// TwinCAT 3 PLC project MotorControl
// ProgramVersion: 3.1.4024.0
// libraries:
//   Tc2_ModbusRTU, * (Beckhoff Automation GmbH)
//   Tc2_Standard, * (Beckhoff Automation GmbH)
//   Tc2_System, * (Beckhoff Automation GmbH)
//   Tc3_Module, * (Beckhoff Automation GmbH)
// project tree:
//   DUTs/ E_Command.TcDUT, E_InverterControlWord.TcDUT, E_InverterStatusWord.TcTLEO, E_InverterError.TcTLEO, E_StateDevice.TcTLEO, ST_Inverter.TcDUT, ST_WorkTime.TcDUT
//   DUTs/Fermentation/ ST_LevelSens.TcDUT, ST_MccRev.TcDUT, ST_PhSens.TcDUT, ST_PressureSens.TcDUT, ST_TempSens.TcDUT
//   GVLs/GVL.FermentationProcess/ Fermentation_001.TcGVL
//   GVLs/ GVL.TcGVL, Itf.TcGVL, Param.TcGVL
//   / PlcTask.TcTTO
//   POUs/Abstraction/ FB_MotorControl.TcPOU, FB_MotorControlInverter.TcPOU, FB_MotorControlReverse.TcPOU
//   POUs/Devices/ Button.TcPOU, Button_1.TcPOU, Contactor.TcPOU, ContactorReverse.TcPOU, NumberEdit.TcPOU, Label.TcPOU, Led.TcPOU, TermFuse.TcPOU
//   POUs/Devices/ITFs/ I_Button.TcIO
//   POUs/Devices/Modbus/ FB_InverterOperation.TcPOU
//   POUs/Implementation/ FB_Drive.TcPOU, FB_DriveInverter.TcPOU, FB_DriveReverse.TcPOU
//   POUs/Implementation/ITFs/ I_Drive.TcIO, I_DriveInverter.TcIO, I_DriveReverse.TcIO
//   POUs/ MAIN.TcPOU, mergeIO.TcPOU
//   POUs/Process/ FermentationProcess_001.TcPOU
//   POUs/Scaling/ FB_Scaling.TcPOU
// (motion and I/O tree: see PLC project mcc)
// real-time tasks:
//   TASK PlcTask2: cycle T#10ms, priority 22, ADS port 352
// variable links:

CONFIGURATION MotorControl
    RESOURCE PLC ON TwinCAT3
        TASK PlcTask(INTERVAL := T#10ms, PRIORITY := 22);
        PROGRAM MAIN WITH PlcTask : MAIN;
    END_RESOURCE
END_CONFIGURATION

// ---- DUTs/E_Command.TcDUT
//{attribute 'qualified_only'}
{attribute 'strict'}
TYPE E_Command :
(
	 eReady, 
	 eFwd, 
	 eRev,
	 eResetInv  
	 
); // domyślna inicjalizacja wszystkich E_ATVCommand Variables na WORD
END_TYPE

// ---- DUTs/E_InverterControlWord.TcDUT
//{attribute 'qualified_only'}
{attribute 'strict'}
TYPE E_InverterControlWord :
(
	 eShutDown         := 16#0006,  //State 2 - Shutdown command -final operating state -> Ready to switch on 
	 eSwitchOn         := 16#0007,  //State 3 - Switch On  command - final operating state -> Switched On Its the same command Disable Operation
	 eEnableOperation  := 16#000F,	//State 4 - Enable Operation - final operating state -> Operation enabled (napęd pracuej do przodu)  
	 eReverseOperation := 16#080F,  //State 4 - Enable Operation Reverse - final operating state -> Operation enabled (napęd pracuej do tyłu)
	 eFaultReset       := 16#0080   //State 5 - Error reset - final operating state -> Ready to switch on 
 	 
)WORD;
END_TYPE

// ---- DUTs/E_InverterStatusWord.TcTLEO
//{attribute 'qualified_only'}
{attribute 'strict'}
TYPE E_InverterStatusWord : // State WORD of ATV Inverter ETA Masked By 0x006f H
(
	eFaultAfterOperation   := 16#0008,	// wykryto błąd po stanie operacyjnym (falownik pracował i nastąpił błąd pracy) po operacji Quick Stop Active przejscie do stanu - 6 falownika
	eFaultDrive            := 16#0028,	// błąd komunikacja Modbus przerwana i nieaktywna SLF1
	eSwitchOnDisabled	   := 16#0040,	// Stan po udanym resecie błędu komunikacji LCD - nSE
	eReadyToSwitchOn       := 16#0021,	// Stan po ustawieniu gotowości Inverta komendą eReady = 14
	eSwitchedOn            := 16#0023,  // Stan po ustawieniu komendy eFwd = 15 lub eRev = 2063 gdy jest zerowa prędkośc zadana speed = 0 
	eOperationEnabled      := 16#0027   // Stan gdy napęd pracuje w kierunku do przodu i do tyłu i osiagnał predkosc zadaną
		
)WORD;
END_TYPE
//  eFaultAfterOperation = '16#0008'
//  eFaultDrive = '16#0028'
//  eSwitchOnDisabled = '16#0040'
//  eReadyToSwitchOn = '16#0021'
//  eSwitchedOn = '16#0023'
//  eOperationEnabled = '16#0027'

// ---- DUTs/E_InverterError.TcTLEO
{attribute 'qualified_only'}
{attribute 'strict'}
TYPE E_InverterError :
(
	nOF := 0,
	InF := 1,
	CFF := 3,
	CFI := 4,
	SLF1:= 5, 
	EPF1:= 8,
	OCF := 9,
	CrF1:= 10,
	OHF := 16,
	OLF := 17,
	ObF := 18,
	OSF := 19,
	OPF1:= 20,
	PHF := 21,
	USF := 22,
	SCF1:= 23,
	SOF := 24,
	tnF := 25,
	InF1:= 26,
	InF2:= 27,
	InF3:= 28,
	InF4:= 29,
	SCF3:= 32,
	OPF2:= 33,
	SLF2:= 42,
	SLF3:= 45,
	InF9:= 51,
	InFb:= 53,
	tJF := 54,
	SCF4:= 55,
	SCF5:= 56,
	InFE:= 69, 
	CFI2:= 77,
	ULF := 100,
	OLC := 101,
	SPIF:= 102,
	LFF1:= 106
	
)WORD;
END_TYPE

// ---- DUTs/E_StateDevice.TcTLEO
//{attribute 'qualified_only'}
{attribute 'strict'}
TYPE E_StateDevice :
(
	eOn       := 0,
	eOff      := 1,
	eForward  := 2,
	eReverse  := 3,
	eReset    := 4,
	eFault    := 5,
	eAuto     := 6
);
END_TYPE

// ---- DUTs/Fermentation/ST_LevelSens.TcDUT
{attribute 'OPC.UA.DA' := '2'}
{attribute 'OPC.UA.DA.StructuredType' := '1'}

TYPE ST_LevelSens :
STRUCT
	
	rRawLevelValue AT%I* : INT;	 // raw value from measure instruments
	rLevelValue  		 : REAL;  // value from fermentation tank Level sensor	

END_STRUCT
END_TYPE

// ---- DUTs/Fermentation/ST_MccRev.TcDUT
{attribute 'OPC.UA.DA' := '2'}
{attribute 'OPC.UA.DA.StructuredType' := '1'}
TYPE ST_MccRev :
STRUCT

	bAutoButton  	   : BOOL;  // SCADA button Auto/manual Command
	bForwardButton     : BOOL;  // SCADA button Forward drive Command
	bReverseButton	   : BOOL;  // SCADA button Reverse drive Command
	bTermFuse    AT%I* : BOOL;  // Term Fuse state from psyhical input
	bContactor   AT%Q* : BOOL;  // Contactor state from psyhical output
	udHours   		   : UDINT; // Work Time Counter - hours nonvolatile memory register
	uMinutes	   	   : UINT;  // Work Time Counter - minuts nonvolatile memory register
	uSeconds           : UINT;  // Work Time Counter - seconds nonvolatile memory register
  	sStatus	           : T_MaxString; // Motor Status string
	sState 	           : T_MaxString; // Motor State string		

END_STRUCT
END_TYPE

// ---- DUTs/Fermentation/ST_PhSens.TcDUT
{attribute 'OPC.UA.DA' := '2'}
{attribute 'OPC.UA.DA.StructuredType' := '1'}

TYPE ST_PhSens :
STRUCT
	
	rRawPhValue AT%I* : INT;	 // raw value from measure instruments
	rPhValue  		  : REAL;    // value from fermentation tank Ph sensor		

END_STRUCT
END_TYPE

// ---- DUTs/Fermentation/ST_PressureSens.TcDUT
{attribute 'OPC.UA.DA' := '2'}
{attribute 'OPC.UA.DA.StructuredType' := '1'}
TYPE ST_PressureSens :
STRUCT
	
	rRawPressureValue AT%I* : INT;	   // raw value from measure instruments
	rPressureValue  		: REAL;    // value from fermentation tank Pressure sensor	

END_STRUCT
END_TYPE

// ---- DUTs/Fermentation/ST_TempSens.TcDUT
{attribute 'OPC.UA.DA' := '2'}
{attribute 'OPC.UA.DA.StructuredType' := '1'}
TYPE ST_TempSens :
STRUCT
	
	rRawTempValue AT%I* : INT;	 // raw value from measure instruments
	rTempValue  		: REAL;  // value from fermentation tank temperature sensor	

END_STRUCT
END_TYPE

// ---- DUTs/ST_Inverter.TcDUT
TYPE ST_Inverter :
STRUCT
	bDeviceId         : BYTE;
	wStatus	          : E_InverterStatusWord;
	eControl          : E_InverterControlWord;
	errorInv  		  : E_InverterError;           // AVT inverter Error
	sErrorDescription : T_MaxString;
	rSpeed	          : WORD;	
	errorMdb          : MODBUS_ERRORS;  // Modbus Communications error		
END_STRUCT
END_TYPE

// ---- DUTs/ST_WorkTime.TcDUT
TYPE ST_WorkTime :
STRUCT
	hours	: UDINT;
	minuts	: UINT;
	seconds	: UINT;
END_STRUCT
END_TYPE

// ---- GVLs/GVL.FermentationProcess/Fermentation_001.TcGVL
{attribute 'qualified_only'}
VAR_GLOBAL
	
	//**************************** Reverse Motor ***************************************************************
	
	{attribute 'OPC.UA.DA' := '1'}
	{attribute 'OPC.UA.DA.StructuredType' := '1'}
	{attribute 'OPC.UA.DA.Description' := 'MccRev (structured) type '} 
	MccRev_001 : ST_MccRev;
	
	{attribute 'OPC.UA.DA' := '1'}
	{attribute 'OPC.UA.DA.StructuredType' := '1'}
	{attribute 'OPC.UA.DA.Description' := 'MccRev (structured) type '} 
	MccRev_002 : ST_MccRev;
	
	{attribute 'OPC.UA.DA' := '1'}
	{attribute 'OPC.UA.DA.StructuredType' := '1'}
	{attribute 'OPC.UA.DA.Description' := 'MccRev (structured) type '} 
	MccRev_003 : ST_MccRev;
	
	{attribute 'OPC.UA.DA' := '1'}
	{attribute 'OPC.UA.DA.StructuredType' := '1'}
	{attribute 'OPC.UA.DA.Description' := 'MccRev (structured) type '} 
	MccRev_004 : ST_MccRev;
	
	{attribute 'OPC.UA.DA' := '1'}
	{attribute 'OPC.UA.DA.StructuredType' := '1'}
	{attribute 'OPC.UA.DA.Description' := 'MccRev (structured) type '} 
	MccRev_005 : ST_MccRev;
	
	{attribute 'OPC.UA.DA' := '1'}
	{attribute 'OPC.UA.DA.StructuredType' := '1'}
	{attribute 'OPC.UA.DA.Description' := 'MccRev (structured) type '} 
	MccRev_006 : ST_MccRev;
	
	{attribute 'OPC.UA.DA' := '1'}
	{attribute 'OPC.UA.DA.StructuredType' := '1'}
	{attribute 'OPC.UA.DA.Description' := 'MccRev (structured) type '} 
	MccRev_007 : ST_MccRev;
	
	{attribute 'OPC.UA.DA' := '1'}
	{attribute 'OPC.UA.DA.StructuredType' := '1'}
	{attribute 'OPC.UA.DA.Description' := 'MccRev (structured) type '} 
	MccRev_008 : ST_MccRev;
	
	{attribute 'OPC.UA.DA' := '1'}
	{attribute 'OPC.UA.DA.StructuredType' := '1'}
	{attribute 'OPC.UA.DA.Description' := 'MccRev (structured) type '} 
	MccRev_009 : ST_MccRev;
	
	{attribute 'OPC.UA.DA' := '1'}
	{attribute 'OPC.UA.DA.StructuredType' := '1'}
	{attribute 'OPC.UA.DA.Description' := 'MccRev (structured) type '} 
	MccRev_010 : ST_MccRev;
	
	{attribute 'OPC.UA.DA' := '1'}
	{attribute 'OPC.UA.DA.StructuredType' := '1'}
	{attribute 'OPC.UA.DA.Description' := 'MccRev (structured) type '} 
	MccRev_011 : ST_MccRev;
	
	
	{attribute 'OPC.UA.DA' := '1'}
	{attribute 'OPC.UA.DA.StructuredType' := '1'}
	{attribute 'OPC.UA.DA.Description' := 'MccRev (structured) type '} 
	MccRev_012 : ST_MccRev;
	
	
	{attribute 'OPC.UA.DA' := '1'}
	{attribute 'OPC.UA.DA.StructuredType' := '1'}
	{attribute 'OPC.UA.DA.Description' := 'MccRev (structured) type '} 
	MccRev_013 : ST_MccRev;
	
	{attribute 'OPC.UA.DA' := '1'}
	{attribute 'OPC.UA.DA.StructuredType' := '1'}
	{attribute 'OPC.UA.DA.Description' := 'MccRev (structured) type '} 
	MccRev_014 : ST_MccRev;
	
	
	{attribute 'OPC.UA.DA' := '1'}
	{attribute 'OPC.UA.DA.StructuredType' := '1'}
	{attribute 'OPC.UA.DA.Description' := 'MccRev (structured) type '} 
	MccRev_015 : ST_MccRev;
	
	
	{attribute 'OPC.UA.DA' := '1'}
	{attribute 'OPC.UA.DA.StructuredType' := '1'}
	{attribute 'OPC.UA.DA.Description' := 'MccRev (structured) type '} 
	MccRev_016 : ST_MccRev;
	
	{attribute 'OPC.UA.DA' := '1'}
	{attribute 'OPC.UA.DA.StructuredType' := '1'}
	{attribute 'OPC.UA.DA.Description' := 'MccRev (structured) type '} 
	MccRev_017 : ST_MccRev;
	
	
	{attribute 'OPC.UA.DA' := '1'}
	{attribute 'OPC.UA.DA.StructuredType' := '1'}
	{attribute 'OPC.UA.DA.Description' := 'MccRev (structured) type '} 
	MccRev_018 : ST_MccRev;
	
	{attribute 'OPC.UA.DA' := '1'}
	{attribute 'OPC.UA.DA.StructuredType' := '1'}
	{attribute 'OPC.UA.DA.Description' := 'MccRev (structured) type '} 
	MccRev_019 : ST_MccRev;
	
	
	{attribute 'OPC.UA.DA' := '1'}
	{attribute 'OPC.UA.DA.StructuredType' := '1'}
	{attribute 'OPC.UA.DA.Description' := 'MccRev (structured) type '} 
	MccRev_020 : ST_MccRev;
	
	
	
	//**************************** Temperature Sensor***************************************************************
	
	{attribute 'OPC.UA.DA' := '1'}
	{attribute 'OPC.UA.DA.AnalogItemType' := '1'}
	{attribute 'OPC.UA.DA.AnalogItemType.EngineeringUnits' := '4408652'  }(*EngeneeringUnit = degree Celsius*)
	{attribute 'OPC.UA.DA.AnalogItemType.InstrumentRange' := '0:100'  }
	{attribute 'OPC.UA.DA.AnalogItemType.EURange' := '53:57'  }
	{attribute 'OPC.UA.DA.AnalogItemType.WriteBehavior' := '2'  } (*AnalogWrMode_AllowAny = 0,
																	AnalogWrMode_Clamp = 1,
																	AnalogWrMode_Reject = 2,*)
	TempSens_001 : ST_TempSens;
	
		//**************************** Temperature Sensor***************************************************************
	
	{attribute 'OPC.UA.DA' := '1'}
	{attribute 'OPC.UA.DA.AnalogItemType' := '1'}
	{attribute 'OPC.UA.DA.AnalogItemType.EngineeringUnits' := '4408652'  }(*EngeneeringUnit = degree Celsius*)
	{attribute 'OPC.UA.DA.AnalogItemType.InstrumentRange' := '0:100'  }
	{attribute 'OPC.UA.DA.AnalogItemType.EURange' := '53:57'  }
	{attribute 'OPC.UA.DA.AnalogItemType.WriteBehavior' := '2'  } (*AnalogWrMode_AllowAny = 0,
																	AnalogWrMode_Clamp = 1,
																	AnalogWrMode_Reject = 2,*)
	TempSens_002 : ST_TempSens;
	
		//**************************** Temperature Sensor***************************************************************
	
	{attribute 'OPC.UA.DA' := '1'}
	{attribute 'OPC.UA.DA.AnalogItemType' := '1'}
	{attribute 'OPC.UA.DA.AnalogItemType.EngineeringUnits' := '4408652'  }(*EngeneeringUnit = degree Celsius*)
	{attribute 'OPC.UA.DA.AnalogItemType.InstrumentRange' := '0:100'  }
	{attribute 'OPC.UA.DA.AnalogItemType.EURange' := '53:57'  }
	{attribute 'OPC.UA.DA.AnalogItemType.WriteBehavior' := '2'  } (*AnalogWrMode_AllowAny = 0,
																	AnalogWrMode_Clamp = 1,
																	AnalogWrMode_Reject = 2,*)
	TempSens_003 : ST_TempSens;
	
	
		//**************************** Level Sensor***************************************************************
			
	{attribute 'OPC.UA.DA' := '1'}
	{attribute 'OPC.UA.DA.AnalogItemType' := '1'}
	{attribute 'OPC.UA.DA.AnalogItemType.EngineeringUnits' := '5067858'  }(*EngeneeringUnit = metre*)
	{attribute 'OPC.UA.DA.AnalogItemType.InstrumentRange' := '0:10'  } (*0- 10m , metry*)
	{attribute 'OPC.UA.DA.AnalogItemType.EURange' := '6:7'  }			(*1m słupa wody to 9,79kPa*)
	{attribute 'OPC.UA.DA.AnalogItemType.WriteBehavior' := '2'  } (*AnalogWrMode_AllowAny = 0,
																	AnalogWrMode_Clamp = 1,
																	AnalogWrMode_Reject = 2,*)
	LevelSens_001 : ST_LevelSens;
																		

		//**************************** Ph Sensor***************************************************************
		
	{attribute 'OPC.UA.DA' := '1'}
	{attribute 'OPC.UA.DA.AnalogItemType' := '1'}
	{attribute 'OPC.UA.DA.AnalogItemType.EngineeringUnits' := '5255734'  }(*EngeneeringUnit = phot*)
	{attribute 'OPC.UA.DA.AnalogItemType.InstrumentRange' := '0:12'  } (*0- 12ph , czujnik od 0 do 12*)
	{attribute 'OPC.UA.DA.AnalogItemType.EURange' := '7:8'  }			(*pracujemy w zakresie od 7 do 8 ph*)
	{attribute 'OPC.UA.DA.AnalogItemType.WriteBehavior' := '2'  } (*AnalogWrMode_AllowAny = 0,
																	AnalogWrMode_Clamp = 1,
																	AnalogWrMode_Reject = 2,*)
	PhSens_001 : ST_PhSens;		
		
		//**************************** Pressure Sensor***************************************************************
		
	{attribute 'OPC.UA.DA' := '1'}
	{attribute 'OPC.UA.DA.AnalogItemType' := '1'}
	{attribute 'OPC.UA.DA.AnalogItemType.EngineeringUnits' := '4935745'  }(*EngeneeringUnit = kPa*)
	{attribute 'OPC.UA.DA.AnalogItemType.InstrumentRange' := '0:5'  } (*0- 5kPa*)
	{attribute 'OPC.UA.DA.AnalogItemType.EURange' := '3:4'  }			(*pracujemy w zakresie od 3 do 4 kPa*)
	{attribute 'OPC.UA.DA.AnalogItemType.WriteBehavior' := '2'  } (*AnalogWrMode_AllowAny = 0,
																	AnalogWrMode_Clamp = 1,
																	AnalogWrMode_Reject = 2,*)
	PressureSens_001 : ST_PressureSens;		
	
	
	
END_VAR

// ---- GVLs/GVL.TcGVL
{attribute 'qualified_only'}
VAR_GLOBAL
	// FB DRIVE MCC_01
	{attribute 'OPC.UA.DA' := '1'}
	bForwardButton_M01     : BOOL;  // SCADA button Forward drive Command 
	bAutoButton_M01  	   : BOOL;  // SCADA button Auto/manual Command
	bAuto_M01			   : BOOL;  // Memory Flag to program execution control  
	bContactor_M01         : BOOL;  // Contactor state from psyhical output
	bTermFuse_M01          : BOOL;  // Term Fuse state from psyhical input
	udHours_M01   		   : UDINT; // Work Time Counter - hours nonvolatile memory register
	uMinuts_M01	   		   : UINT;  // Work Time Counter - minuts nonvolatile memory register
	uSeconds_M01           : UINT;  // Work Time Counter - seconds nonvolatile memory register
  	sStatus_M01	           : T_MaxString; // Motor Status string
	sState_M01 	           : T_MaxString; // Motor State string

END_VAR

{attribute 'qualified_only'}
VAR_GLOBAL
	//FB Drive Inverter MCC_02
	{attribute 'OPC.UA.DA' := '1'}
	bForwardButton_M02     : BOOL;  // SCADA button Forward drive Command 
	bReverseButton_M02     : BOOL;  // SCADA button Reverse drive Command
	bResetButton_M02	   : BOOL;  // SCADA button Reset drive Command
	bAutoButton_M02  	   : BOOL;  // SCADA button Auto/manual Command
	rSpeedEdit_M02		   : REAL;	// SCADA textEdit Speed value
	bAuto_M02			   : BOOL;  // Memory Flag to program execution control  
	bTermFuse_M02          : BOOL;  // Term Fuse state from psyhical input
	udHours_M02   		   : UDINT; // Work Time Counter - hours nonvolatile memory register
	uMinuts_M02	   		   : UINT;  // Work Time Counter - minuts nonvolatile memory register
	uSeconds_M02           : UINT;  // Work Time Counter - seconds nonvolatile memory register
  	sStatus_M02	           : T_MaxString; // Motor Status string
	sState_M02 	           : T_MaxString; // Motor State string	
END_VAR

// ---- GVLs/Itf.TcGVL
{attribute 'qualified_only'}
VAR_GLOBAL
	
	
	aItfDriveInverter		  : ARRAY [1..Param.cMaxInverter] OF I_DriveInverter; // Array of Interface variable
	
END_VAR

// ---- GVLs/Param.TcGVL
{attribute 'qualified_only'}
VAR_GLOBAL CONSTANT
	// size of max AVT inverter in network Modbus RTU
	cMaxInverter	: INT := 31;
END_VAR

// ---- POUs/Devices/ITFs/I_Button.TcIO
INTERFACE I_Button

PROPERTY IsPressed : BOOL
GET
END_GET
SET
END_SET
END_PROPERTY

END_INTERFACE

// ---- POUs/Implementation/ITFs/I_Drive.TcIO
INTERFACE I_Drive EXTENDS __SYSTEM.IQueryInterface

METHOD AutoLedOff : BOOL
VAR_INPUT
END_VAR
END_METHOD

METHOD AutoLedOn : BOOL
VAR_INPUT
END_VAR
END_METHOD

PROPERTY Hours : UDINT
GET
END_GET
SET
END_SET
END_PROPERTY

PROPERTY Minuts : UINT
GET
END_GET
SET
END_SET
END_PROPERTY

PROPERTY MotorAuto : BOOL
GET
END_GET
SET
END_SET
END_PROPERTY

PROPERTY MotorProtection : BOOL
GET
END_GET
END_PROPERTY

PROPERTY MotorState : T_MaxString
GET
END_GET
SET
END_SET
END_PROPERTY

PROPERTY MotorStatus : T_MaxString
GET
END_GET
SET
END_SET
END_PROPERTY

PROPERTY MotorSupply : BOOL
GET
END_GET
END_PROPERTY

PROPERTY Seconds : UINT
GET
END_GET
SET
END_SET
END_PROPERTY

METHOD StatusState : E_StateDevice
VAR_INPUT
END_VAR
END_METHOD

METHOD SwitchOff : BOOL
VAR_INPUT
END_VAR
END_METHOD

METHOD SwitchOn : BOOL
VAR_INPUT
END_VAR
END_METHOD

METHOD PUBLIC WorkCount : STRING
VAR_INPUT
END_VAR
END_METHOD

METHOD WorkCounterOff : BOOL
VAR_INPUT
	
END_VAR
END_METHOD

METHOD WorkCounterOn : BOOL
VAR_INPUT

END_VAR
END_METHOD

END_INTERFACE

// ---- POUs/Implementation/ITFs/I_DriveInverter.TcIO
INTERFACE I_DriveInverter EXTENDS I_DriveReverse

PROPERTY DeviceData : ST_Inverter
GET
END_GET
SET
END_SET
END_PROPERTY

PROPERTY InstanceCounter : INT
GET
END_GET
END_PROPERTY

METHOD Reset : BOOL
VAR_INPUT
END_VAR
END_METHOD

METHOD SetSpeed : BOOL
VAR_INPUT
	_speed : REAL;
END_VAR
END_METHOD

END_INTERFACE

// ---- POUs/Implementation/ITFs/I_DriveReverse.TcIO
INTERFACE I_DriveReverse EXTENDS I_Drive

METHOD SwitchReverseOff : BOOL
VAR_INPUT
END_VAR
END_METHOD

METHOD SwitchReverseON : BOOL
VAR_INPUT
END_VAR
END_METHOD

END_INTERFACE

// ---- POUs/MAIN.TcPOU
PROGRAM MAIN
VAR
	
	// Drive
	//fbDrive			          : FB_Drive;
	//fbDriveReverse	          : FB_DriveReverse;
	//bUnitId              	  : BYTE:=1; //adres napędu falownikowego Higienizatora
	
	//fbDriveInverter1		  : FB_DriveInverter(1);
	//fbDriveInverter2		  : FB_DriveInverter(2);

	//Drive Control	
//	fbMotorControl_001 	     	  : FB_MotorControl(fbDrive);
//	fbMotorControl_002 	     	  : FB_MotorControl(fbDrive);
	
	//fbMotorControlReverse_001 	  : FB_MotorControlReverse(fbDriveReverse);
	//fbMotorControlReverse_001 	  : FB_MotorControlReverse(fbDriveReverse);
	
	
	//fbMotorControlInverter    : FB_MotorControlInverter(fbDriveInverter1);
	
//fbMotorControlInverter2    : FB_MotorControlInverter(fbDriveInverter2);	
	
	{attribute 'OPC.UA.DA' := '1'}
	rReal3 : REAL;

	//Modbus RTU - obiektów tej klasy może być tylko tyle ile jest dostępnych fizycznych portów RS485
	//np. dla modułu EL6022 są dwa fizyczne porty RS485
	//fbInverterOperation		   : FB_InverterOperation;
	


	
END_VAR

//Ustaw zmienne SCADY i PLC
//mergeIO();

//Processy
FermentationProcess_001();








//Fermentation Process
//fbMotorControlReverse();


//fbMotorControlInverter();
//fbMotorControlInverter2();
//fbInverterOperation();

END_PROGRAM

// ---- POUs/Process/FermentationProcess_001.TcPOU
PROGRAM FermentationProcess_001
VAR
	

	//MCC Driver	
	fbDriveReverse_001		      : FB_DriveReverse;
	fbDriveReverse_002		      : FB_DriveReverse;
	fbDriveReverse_003		      : FB_DriveReverse;
	fbDriveReverse_004		      : FB_DriveReverse;
	fbDriveReverse_005		      : FB_DriveReverse;
	fbDriveReverse_006		      : FB_DriveReverse;
	fbDriveReverse_007		      : FB_DriveReverse;
	fbDriveReverse_008		      : FB_DriveReverse;
	fbDriveReverse_009		      : FB_DriveReverse;
	fbDriveReverse_010		      : FB_DriveReverse;
	fbDriveReverse_011		      : FB_DriveReverse;
	fbDriveReverse_012		      : FB_DriveReverse;
	fbDriveReverse_013		      : FB_DriveReverse;
	fbDriveReverse_014		      : FB_DriveReverse;
	fbDriveReverse_015		      : FB_DriveReverse;
	fbDriveReverse_016		      : FB_DriveReverse;
	fbDriveReverse_017		      : FB_DriveReverse;
	fbDriveReverse_018		      : FB_DriveReverse;
	fbDriveReverse_019		      : FB_DriveReverse;
	fbDriveReverse_020		      : FB_DriveReverse;


	//MCC Driver Control
	fbMccRev_001			 	  : FB_MotorControlReverse(fbDriveReverse_001);
	fbMccRev_002			 	  : FB_MotorControlReverse(fbDriveReverse_002);
	fbMccRev_003			 	  : FB_MotorControlReverse(fbDriveReverse_003);
	fbMccRev_004 	 			  : FB_MotorControlReverse(fbDriveReverse_004);
	fbMccRev_005			 	  : FB_MotorControlReverse(fbDriveReverse_005);
	fbMccRev_006			 	  : FB_MotorControlReverse(fbDriveReverse_006);
	fbMccRev_007				  : FB_MotorControlReverse(fbDriveReverse_007);
	fbMccRev_008 	 			  : FB_MotorControlReverse(fbDriveReverse_008);
	fbMccRev_009 	  			  : FB_MotorControlReverse(fbDriveReverse_009);
	fbMccRev_010 	              : FB_MotorControlReverse(fbDriveReverse_010);
	fbMccRev_011			 	  : FB_MotorControlReverse(fbDriveReverse_011);
	fbMccRev_012			 	  : FB_MotorControlReverse(fbDriveReverse_012);
	fbMccRev_013			 	  : FB_MotorControlReverse(fbDriveReverse_013);
	fbMccRev_014 	 			  : FB_MotorControlReverse(fbDriveReverse_014);
	fbMccRev_015			 	  : FB_MotorControlReverse(fbDriveReverse_015);
	fbMccRev_016			 	  : FB_MotorControlReverse(fbDriveReverse_016);
	fbMccRev_017				  : FB_MotorControlReverse(fbDriveReverse_017);
	fbMccRev_018 	 			  : FB_MotorControlReverse(fbDriveReverse_018);
	fbMccRev_019 	  			  : FB_MotorControlReverse(fbDriveReverse_019);
	fbMccRev_020 	              : FB_MotorControlReverse(fbDriveReverse_020);
	
	//Temperature Sensor
	fbTempSens_001				  : FB_Scaling;
	fbTempSens_002				  : FB_Scaling;
	fbTempSens_003				  : FB_Scaling;
	//Level Sensor
	fbLevelSens_001				  : FB_Scaling;
	//Ph Sensor
	fbPhSens_001				  : FB_Scaling;	
	//Pressure Sensor
	fbPressureSens_001			  : FB_Scaling;	
	
	
	
	
	
END_VAR

ACT_Motor();
ACT_TempSens();
ACT_LevelSens();
ACT_PhSens();

ACTION ACT_LevelSens:
fbLevelSens_001(
    _rX := Fermentation_001.LevelSens_001.rRawLevelValue,
    _rXmin := 0,
    _rXmax := 32767,
    _rYmin := 0,
    _rYmax := 100); // FB_Scaling
Fermentation_001.LevelSens_001.rLevelValue := fbLevelSens_001._rY;
END_ACTION

ACTION ACT_Motor:
//Sygnały obiektów MccRev_* mieszadeł fermentora

//***************************************************SCADA********************************************************

//MccRev_001 variable sets by SCADA
FermentationProcess_001.fbMccRev_001.ScadaAutoButton     := Fermentation_001.MccRev_001.bAutoButton;    // SCADA button Auto Command
FermentationProcess_001.fbMccRev_001.ScadaForwardButton  := Fermentation_001.MccRev_001.bForwardButton; // SCADA button Forward Command
FermentationProcess_001.fbMccRev_001.ScadaReverseButton  := Fermentation_001.MccRev_001.bReverseButton; // SCADA button Reverse Command

//MccRev_002 variable sets by SCADA
FermentationProcess_001.fbMccRev_002.ScadaAutoButton     := Fermentation_001.MccRev_002.bAutoButton;    // SCADA button Auto Command
FermentationProcess_001.fbMccRev_002.ScadaForwardButton  := Fermentation_001.MccRev_002.bForwardButton; // SCADA button Forward Command
FermentationProcess_001.fbMccRev_002.ScadaReverseButton  := Fermentation_001.MccRev_002.bReverseButton; // SCADA button Reverse Command

//MccRev_003 variable sets by SCADA
FermentationProcess_001.fbMccRev_003.ScadaAutoButton     := Fermentation_001.MccRev_003.bAutoButton;    // SCADA button Auto Command
FermentationProcess_001.fbMccRev_003.ScadaForwardButton  := Fermentation_001.MccRev_003.bForwardButton; // SCADA button Forward Command
FermentationProcess_001.fbMccRev_003.ScadaReverseButton  := Fermentation_001.MccRev_003.bReverseButton; // SCADA button Reverse Command

//MccRev_004 variable sets by SCADA
FermentationProcess_001.fbMccRev_004.ScadaAutoButton     := Fermentation_001.MccRev_004.bAutoButton;    // SCADA button Auto Command
FermentationProcess_001.fbMccRev_004.ScadaForwardButton  := Fermentation_001.MccRev_004.bForwardButton; // SCADA button Forward Command
FermentationProcess_001.fbMccRev_004.ScadaReverseButton  := Fermentation_001.MccRev_004.bReverseButton; // SCADA button Reverse Command

//MccRev_005 variable sets by SCADA
FermentationProcess_001.fbMccRev_005.ScadaAutoButton     := Fermentation_001.MccRev_005.bAutoButton;    // SCADA button Auto Command
FermentationProcess_001.fbMccRev_005.ScadaForwardButton  := Fermentation_001.MccRev_005.bForwardButton; // SCADA button Forward Command
FermentationProcess_001.fbMccRev_005.ScadaReverseButton  := Fermentation_001.MccRev_005.bReverseButton; // SCADA button Reverse Command

//MccRev_006 variable sets by SCADA
FermentationProcess_001.fbMccRev_006.ScadaAutoButton     := Fermentation_001.MccRev_006.bAutoButton;    // SCADA button Auto Command
FermentationProcess_001.fbMccRev_006.ScadaForwardButton  := Fermentation_001.MccRev_006.bForwardButton; // SCADA button Forward Command
FermentationProcess_001.fbMccRev_006.ScadaReverseButton  := Fermentation_001.MccRev_006.bReverseButton; // SCADA button Reverse Command

//MccRev_007 variable sets by SCADA
FermentationProcess_001.fbMccRev_007.ScadaAutoButton     := Fermentation_001.MccRev_007.bAutoButton;    // SCADA button Auto Command
FermentationProcess_001.fbMccRev_007.ScadaForwardButton  := Fermentation_001.MccRev_007.bForwardButton; // SCADA button Forward Command
FermentationProcess_001.fbMccRev_007.ScadaReverseButton  := Fermentation_001.MccRev_007.bReverseButton; // SCADA button Reverse Command

//MccRev_008 variable sets by SCADA
FermentationProcess_001.fbMccRev_008.ScadaAutoButton     := Fermentation_001.MccRev_008.bAutoButton;    // SCADA button Auto Command
FermentationProcess_001.fbMccRev_008.ScadaForwardButton  := Fermentation_001.MccRev_008.bForwardButton; // SCADA button Forward Command
FermentationProcess_001.fbMccRev_008.ScadaReverseButton  := Fermentation_001.MccRev_008.bReverseButton; // SCADA button Reverse Command

//MccRev_009 variable sets by SCADA
FermentationProcess_001.fbMccRev_009.ScadaAutoButton     := Fermentation_001.MccRev_009.bAutoButton;    // SCADA button Auto Command
FermentationProcess_001.fbMccRev_009.ScadaForwardButton  := Fermentation_001.MccRev_009.bForwardButton; // SCADA button Forward Command
FermentationProcess_001.fbMccRev_009.ScadaReverseButton  := Fermentation_001.MccRev_009.bReverseButton; // SCADA button Reverse Command

//MccRev_010 variable sets by SCADA
FermentationProcess_001.fbMccRev_010.ScadaAutoButton     := Fermentation_001.MccRev_010.bAutoButton;    // SCADA button Auto Command
FermentationProcess_001.fbMccRev_010.ScadaForwardButton  := Fermentation_001.MccRev_010.bForwardButton; // SCADA button Forward Command
FermentationProcess_001.fbMccRev_010.ScadaReverseButton  := Fermentation_001.MccRev_010.bReverseButton; // SCADA button Reverse Command

//MccRev_011 variable sets by SCADA
FermentationProcess_001.fbMccRev_011.ScadaAutoButton     := Fermentation_001.MccRev_011.bAutoButton;    // SCADA button Auto Command
FermentationProcess_001.fbMccRev_011.ScadaForwardButton  := Fermentation_001.MccRev_011.bForwardButton; // SCADA button Forward Command
FermentationProcess_001.fbMccRev_011.ScadaReverseButton  := Fermentation_001.MccRev_011.bReverseButton; // SCADA button Reverse Command

//MccRev_012 variable sets by SCADA
FermentationProcess_001.fbMccRev_012.ScadaAutoButton     := Fermentation_001.MccRev_012.bAutoButton;    // SCADA button Auto Command
FermentationProcess_001.fbMccRev_012.ScadaForwardButton  := Fermentation_001.MccRev_012.bForwardButton; // SCADA button Forward Command
FermentationProcess_001.fbMccRev_012.ScadaReverseButton  := Fermentation_001.MccRev_012.bReverseButton; // SCADA button Reverse Command

//MccRev_013 variable sets by SCADA
FermentationProcess_001.fbMccRev_013.ScadaAutoButton     := Fermentation_001.MccRev_013.bAutoButton;    // SCADA button Auto Command
FermentationProcess_001.fbMccRev_013.ScadaForwardButton  := Fermentation_001.MccRev_013.bForwardButton; // SCADA button Forward Command
FermentationProcess_001.fbMccRev_013.ScadaReverseButton  := Fermentation_001.MccRev_013.bReverseButton; // SCADA button Reverse Command

//MccRev_014 variable sets by SCADA
FermentationProcess_001.fbMccRev_014.ScadaAutoButton     := Fermentation_001.MccRev_014.bAutoButton;    // SCADA button Auto Command
FermentationProcess_001.fbMccRev_014.ScadaForwardButton  := Fermentation_001.MccRev_014.bForwardButton; // SCADA button Forward Command
FermentationProcess_001.fbMccRev_014.ScadaReverseButton  := Fermentation_001.MccRev_014.bReverseButton; // SCADA button Reverse Command

//MccRev_015 variable sets by SCADA
FermentationProcess_001.fbMccRev_015.ScadaAutoButton     := Fermentation_001.MccRev_015.bAutoButton;    // SCADA button Auto Command
FermentationProcess_001.fbMccRev_015.ScadaForwardButton  := Fermentation_001.MccRev_015.bForwardButton; // SCADA button Forward Command
FermentationProcess_001.fbMccRev_015.ScadaReverseButton  := Fermentation_001.MccRev_015.bReverseButton; // SCADA button Reverse Command

//MccRev_016 variable sets by SCADA
FermentationProcess_001.fbMccRev_016.ScadaAutoButton     := Fermentation_001.MccRev_016.bAutoButton;    // SCADA button Auto Command
FermentationProcess_001.fbMccRev_016.ScadaForwardButton  := Fermentation_001.MccRev_016.bForwardButton; // SCADA button Forward Command
FermentationProcess_001.fbMccRev_016.ScadaReverseButton  := Fermentation_001.MccRev_016.bReverseButton; // SCADA button Reverse Command

//MccRev_017 variable sets by SCADA
FermentationProcess_001.fbMccRev_017.ScadaAutoButton     := Fermentation_001.MccRev_017.bAutoButton;    // SCADA button Auto Command
FermentationProcess_001.fbMccRev_017.ScadaForwardButton  := Fermentation_001.MccRev_017.bForwardButton; // SCADA button Forward Command
FermentationProcess_001.fbMccRev_017.ScadaReverseButton  := Fermentation_001.MccRev_017.bReverseButton; // SCADA button Reverse Command

//MccRev_018 variable sets by SCADA
FermentationProcess_001.fbMccRev_018.ScadaAutoButton     := Fermentation_001.MccRev_018.bAutoButton;    // SCADA button Auto Command
FermentationProcess_001.fbMccRev_018.ScadaForwardButton  := Fermentation_001.MccRev_018.bForwardButton; // SCADA button Forward Command
FermentationProcess_001.fbMccRev_018.ScadaReverseButton  := Fermentation_001.MccRev_018.bReverseButton; // SCADA button Reverse Command

//MccRev_019 variable sets by SCADA
FermentationProcess_001.fbMccRev_019.ScadaAutoButton     := Fermentation_001.MccRev_019.bAutoButton;    // SCADA button Auto Command
FermentationProcess_001.fbMccRev_019.ScadaForwardButton  := Fermentation_001.MccRev_019.bForwardButton; // SCADA button Forward Command
FermentationProcess_001.fbMccRev_019.ScadaReverseButton  := Fermentation_001.MccRev_019.bReverseButton; // SCADA button Reverse Command

//MccRev_020 variable sets by SCADA
FermentationProcess_001.fbMccRev_020.ScadaAutoButton     := Fermentation_001.MccRev_020.bAutoButton;    // SCADA button Auto Command
FermentationProcess_001.fbMccRev_020.ScadaForwardButton  := Fermentation_001.MccRev_020.bForwardButton; // SCADA button Forward Command
FermentationProcess_001.fbMccRev_020.ScadaReverseButton  := Fermentation_001.MccRev_020.bReverseButton; // SCADA button Reverse Command


//***************************************************PLC********************************************************************


//MccRev_001 variable sets by PLC
FermentationProcess_001.fbDriveReverse_001.MotorProtection := Fermentation_001.MccRev_001.bTermFuse;       // PLC input thermal fuse
Fermentation_001.MccRev_001.bContactor     := FermentationProcess_001.fbDriveReverse_001.MotorContactor;   // PLC output contactor
Fermentation_001.MccRev_001.udHours        := FermentationProcess_001.fbDriveReverse_001.Hours;            // PLC Work Time Counter - hours nonvolatile memory register
Fermentation_001.MccRev_001.uMinutes       := FermentationProcess_001.fbDriveReverse_001.Minuts;           // PLC Work Time Counter - minutes nonvolatile memory register
Fermentation_001.MccRev_001.uSeconds       := FermentationProcess_001.fbDriveReverse_001.Seconds;          // PLC Work Time Counter - seconds nonvolatile memory register
Fermentation_001.MccRev_001.sState         := FermentationProcess_001.fbDriveReverse_001.MotorState;       // PLC Work Time Counter - minutes nonvolatile memory register
Fermentation_001.MccRev_001.sStatus        := FermentationProcess_001.fbDriveReverse_001.MotorStatus;      // PLC Work Time Counter - seconds nonvolatile memory register


//MccRev_002 variable sets by PLC
FermentationProcess_001.fbDriveReverse_002.MotorProtection := Fermentation_001.MccRev_002.bTermFuse;       // PLC input thermal fuse
Fermentation_001.MccRev_002.bContactor     := FermentationProcess_001.fbDriveReverse_002.MotorContactor;   // PLC output contactor
Fermentation_001.MccRev_002.udHours        := FermentationProcess_001.fbDriveReverse_002.Hours;            // PLC Work Time Counter - hours nonvolatile memory register
Fermentation_001.MccRev_002.uMinutes       := FermentationProcess_001.fbDriveReverse_002.Minuts;           // PLC Work Time Counter - minutes nonvolatile memory register
Fermentation_001.MccRev_002.uSeconds       := FermentationProcess_001.fbDriveReverse_002.Seconds;          // PLC Work Time Counter - seconds nonvolatile memory register
Fermentation_001.MccRev_002.sState         := FermentationProcess_001.fbDriveReverse_002.MotorState;       // PLC Work Time Counter - minutes nonvolatile memory register
Fermentation_001.MccRev_002.sStatus        := FermentationProcess_001.fbDriveReverse_002.MotorStatus;      // PLC Work Time Counter - seconds nonvolatile memory register

//MccRev_003 variable sets by PLC
FermentationProcess_001.fbDriveReverse_003.MotorProtection :=Fermentation_001.MccRev_003.bTermFuse;       // PLC input thermal fuse
Fermentation_001.MccRev_003.bContactor     := FermentationProcess_001.fbDriveReverse_003.MotorContactor;   // PLC output contactor
Fermentation_001.MccRev_003.udHours        := FermentationProcess_001.fbDriveReverse_003.Hours;            // PLC Work Time Counter - hours nonvolatile memory register
Fermentation_001.MccRev_003.uMinutes       := FermentationProcess_001.fbDriveReverse_003.Minuts;           // PLC Work Time Counter - minutes nonvolatile memory register
Fermentation_001.MccRev_003.uSeconds       := FermentationProcess_001.fbDriveReverse_003.Seconds;          // PLC Work Time Counter - seconds nonvolatile memory register
Fermentation_001.MccRev_003.sState         := FermentationProcess_001.fbDriveReverse_003.MotorState;       // PLC Work Time Counter - minutes nonvolatile memory register
Fermentation_001.MccRev_003.sStatus        := FermentationProcess_001.fbDriveReverse_003.MotorStatus;      // PLC Work Time Counter - seconds nonvolatile memory register

//MccRev_004 variable sets by PLC
FermentationProcess_001.fbDriveReverse_004.MotorProtection := Fermentation_001.MccRev_004.bTermFuse;       // PLC input thermal fuse
Fermentation_001.MccRev_004.bContactor     := FermentationProcess_001.fbDriveReverse_004.MotorContactor;   // PLC output contactor
Fermentation_001.MccRev_004.udHours        := FermentationProcess_001.fbDriveReverse_004.Hours;            // PLC Work Time Counter - hours nonvolatile memory register
Fermentation_001.MccRev_004.uMinutes       := FermentationProcess_001.fbDriveReverse_004.Minuts;           // PLC Work Time Counter - minutes nonvolatile memory register
Fermentation_001.MccRev_004.uSeconds       := FermentationProcess_001.fbDriveReverse_004.Seconds;          // PLC Work Time Counter - seconds nonvolatile memory register
Fermentation_001.MccRev_004.sState         := FermentationProcess_001.fbDriveReverse_004.MotorState;       // PLC Work Time Counter - minutes nonvolatile memory register
Fermentation_001.MccRev_004.sStatus        := FermentationProcess_001.fbDriveReverse_004.MotorStatus;      // PLC Work Time Counter - seconds nonvolatile memory register


//MccRev_005 variable sets by PLC
FermentationProcess_001.fbDriveReverse_005.MotorProtection := Fermentation_001.MccRev_005.bTermFuse;       // PLC input thermal fuse
Fermentation_001.MccRev_005.bContactor     := FermentationProcess_001.fbDriveReverse_005.MotorContactor;   // PLC output contactor
Fermentation_001.MccRev_005.udHours        := FermentationProcess_001.fbDriveReverse_005.Hours;            // PLC Work Time Counter - hours nonvolatile memory register
Fermentation_001.MccRev_005.uMinutes       := FermentationProcess_001.fbDriveReverse_005.Minuts;           // PLC Work Time Counter - minutes nonvolatile memory register
Fermentation_001.MccRev_005.uSeconds       := FermentationProcess_001.fbDriveReverse_005.Seconds;          // PLC Work Time Counter - seconds nonvolatile memory register
Fermentation_001.MccRev_005.sState         := FermentationProcess_001.fbDriveReverse_005.MotorState;       // PLC Work Time Counter - minutes nonvolatile memory register
Fermentation_001.MccRev_005.sStatus        := FermentationProcess_001.fbDriveReverse_005.MotorStatus;      // PLC Work Time Counter - seconds nonvolatile memory register


//MccRev_006 variable sets by PLC
FermentationProcess_001.fbDriveReverse_006.MotorProtection := Fermentation_001.MccRev_006.bTermFuse;       // PLC input thermal fuse
Fermentation_001.MccRev_006.bContactor     := FermentationProcess_001.fbDriveReverse_006.MotorContactor;   // PLC output contactor
Fermentation_001.MccRev_006.udHours        := FermentationProcess_001.fbDriveReverse_006.Hours;            // PLC Work Time Counter - hours nonvolatile memory register
Fermentation_001.MccRev_006.uMinutes       := FermentationProcess_001.fbDriveReverse_006.Minuts;           // PLC Work Time Counter - minutes nonvolatile memory register
Fermentation_001.MccRev_006.uSeconds       := FermentationProcess_001.fbDriveReverse_006.Seconds;          // PLC Work Time Counter - seconds nonvolatile memory register
Fermentation_001.MccRev_006.sState         := FermentationProcess_001.fbDriveReverse_006.MotorState;       // PLC Work Time Counter - minutes nonvolatile memory register
Fermentation_001.MccRev_006.sStatus        := FermentationProcess_001.fbDriveReverse_006.MotorStatus;      // PLC Work Time Counter - seconds nonvolatile memory register

//MccRev_007 variable sets by PLC
FermentationProcess_001.fbDriveReverse_007.MotorProtection := Fermentation_001.MccRev_007.bTermFuse;       // PLC input thermal fuse
Fermentation_001.MccRev_007.bContactor     := FermentationProcess_001.fbDriveReverse_007.MotorContactor;   // PLC output contactor
Fermentation_001.MccRev_007.udHours        := FermentationProcess_001.fbDriveReverse_007.Hours;            // PLC Work Time Counter - hours nonvolatile memory register
Fermentation_001.MccRev_007.uMinutes       := FermentationProcess_001.fbDriveReverse_007.Minuts;           // PLC Work Time Counter - minutes nonvolatile memory register
Fermentation_001.MccRev_007.uSeconds       := FermentationProcess_001.fbDriveReverse_007.Seconds;          // PLC Work Time Counter - seconds nonvolatile memory register
Fermentation_001.MccRev_007.sState         := FermentationProcess_001.fbDriveReverse_007.MotorState;       // PLC Work Time Counter - minutes nonvolatile memory register
Fermentation_001.MccRev_007.sStatus        := FermentationProcess_001.fbDriveReverse_007.MotorStatus;      // PLC Work Time Counter - seconds nonvolatile memory register

//MccRev_008 variable sets by PLC
FermentationProcess_001.fbDriveReverse_008.MotorProtection := Fermentation_001.MccRev_008.bTermFuse;       // PLC input thermal fuse
Fermentation_001.MccRev_008.bContactor     := FermentationProcess_001.fbDriveReverse_008.MotorContactor;   // PLC output contactor
Fermentation_001.MccRev_008.udHours        := FermentationProcess_001.fbDriveReverse_008.Hours;            // PLC Work Time Counter - hours nonvolatile memory register
Fermentation_001.MccRev_008.uMinutes       := FermentationProcess_001.fbDriveReverse_008.Minuts;           // PLC Work Time Counter - minutes nonvolatile memory register
Fermentation_001.MccRev_008.uSeconds       := FermentationProcess_001.fbDriveReverse_008.Seconds;          // PLC Work Time Counter - seconds nonvolatile memory register
Fermentation_001.MccRev_008.sState         := FermentationProcess_001.fbDriveReverse_008.MotorState;       // PLC Work Time Counter - minutes nonvolatile memory register
Fermentation_001.MccRev_008.sStatus        := FermentationProcess_001.fbDriveReverse_008.MotorStatus;      // PLC Work Time Counter - seconds nonvolatile memory register


//MccRev_009 variable sets by PLC
FermentationProcess_001.fbDriveReverse_009.MotorProtection := Fermentation_001.MccRev_009.bTermFuse;       // PLC input thermal fuse
Fermentation_001.MccRev_009.bContactor     := FermentationProcess_001.fbDriveReverse_009.MotorContactor;   // PLC output contactor
Fermentation_001.MccRev_009.udHours        := FermentationProcess_001.fbDriveReverse_009.Hours;            // PLC Work Time Counter - hours nonvolatile memory register
Fermentation_001.MccRev_009.uMinutes       := FermentationProcess_001.fbDriveReverse_009.Minuts;           // PLC Work Time Counter - minutes nonvolatile memory register
Fermentation_001.MccRev_009.uSeconds       := FermentationProcess_001.fbDriveReverse_009.Seconds;          // PLC Work Time Counter - seconds nonvolatile memory register
Fermentation_001.MccRev_009.sState         := FermentationProcess_001.fbDriveReverse_009.MotorState;       // PLC Work Time Counter - minutes nonvolatile memory register
Fermentation_001.MccRev_009.sStatus        := FermentationProcess_001.fbDriveReverse_009.MotorStatus;      // PLC Work Time Counter - seconds nonvolatile memory register

//MccRev_010 variable sets by PLC
FermentationProcess_001.fbDriveReverse_010.MotorProtection := Fermentation_001.MccRev_010.bTermFuse;       // PLC input thermal fuse
Fermentation_001.MccRev_010.bContactor     := FermentationProcess_001.fbDriveReverse_010.MotorContactor;   // PLC output contactor
Fermentation_001.MccRev_010.udHours        := FermentationProcess_001.fbDriveReverse_010.Hours;            // PLC Work Time Counter - hours nonvolatile memory register
Fermentation_001.MccRev_010.uMinutes       := FermentationProcess_001.fbDriveReverse_010.Minuts;           // PLC Work Time Counter - minutes nonvolatile memory register
Fermentation_001.MccRev_010.uSeconds       := FermentationProcess_001.fbDriveReverse_010.Seconds;          // PLC Work Time Counter - seconds nonvolatile memory register
Fermentation_001.MccRev_010.sState         := FermentationProcess_001.fbDriveReverse_010.MotorState;       // PLC Work Time Counter - minutes nonvolatile memory register
Fermentation_001.MccRev_010.sStatus        := FermentationProcess_001.fbDriveReverse_010.MotorStatus;      // PLC Work Time Counter - seconds nonvolatile memory register

//MccRev_011 variable sets by PLC
FermentationProcess_001.fbDriveReverse_011.MotorProtection := Fermentation_001.MccRev_011.bTermFuse;       // PLC input thermal fuse
Fermentation_001.MccRev_011.bContactor     := FermentationProcess_001.fbDriveReverse_011.MotorContactor;   // PLC output contactor
Fermentation_001.MccRev_011.udHours        := FermentationProcess_001.fbDriveReverse_011.Hours;            // PLC Work Time Counter - hours nonvolatile memory register
Fermentation_001.MccRev_011.uMinutes       := FermentationProcess_001.fbDriveReverse_011.Minuts;           // PLC Work Time Counter - minutes nonvolatile memory register
Fermentation_001.MccRev_011.uSeconds       := FermentationProcess_001.fbDriveReverse_011.Seconds;          // PLC Work Time Counter - seconds nonvolatile memory register
Fermentation_001.MccRev_011.sState         := FermentationProcess_001.fbDriveReverse_011.MotorState;       // PLC Work Time Counter - minutes nonvolatile memory register
Fermentation_001.MccRev_011.sStatus        := FermentationProcess_001.fbDriveReverse_011.MotorStatus;      // PLC Work Time Counter - seconds nonvolatile memory register


//MccRev_012 variable sets by PLC
FermentationProcess_001.fbDriveReverse_012.MotorProtection := Fermentation_001.MccRev_012.bTermFuse;       // PLC input thermal fuse
Fermentation_001.MccRev_012.bContactor     := FermentationProcess_001.fbDriveReverse_012.MotorContactor;   // PLC output contactor
Fermentation_001.MccRev_012.udHours        := FermentationProcess_001.fbDriveReverse_012.Hours;            // PLC Work Time Counter - hours nonvolatile memory register
Fermentation_001.MccRev_012.uMinutes       := FermentationProcess_001.fbDriveReverse_012.Minuts;           // PLC Work Time Counter - minutes nonvolatile memory register
Fermentation_001.MccRev_012.uSeconds       := FermentationProcess_001.fbDriveReverse_012.Seconds;          // PLC Work Time Counter - seconds nonvolatile memory register
Fermentation_001.MccRev_012.sState         := FermentationProcess_001.fbDriveReverse_012.MotorState;       // PLC Work Time Counter - minutes nonvolatile memory register
Fermentation_001.MccRev_012.sStatus        := FermentationProcess_001.fbDriveReverse_012.MotorStatus;      // PLC Work Time Counter - seconds nonvolatile memory register


//MccRev_013 variable sets by PLC
FermentationProcess_001.fbDriveReverse_013.MotorProtection := Fermentation_001.MccRev_013.bTermFuse;       // PLC input thermal fuse
Fermentation_001.MccRev_013.bContactor     := FermentationProcess_001.fbDriveReverse_013.MotorContactor;   // PLC output contactor
Fermentation_001.MccRev_013.udHours        := FermentationProcess_001.fbDriveReverse_013.Hours;            // PLC Work Time Counter - hours nonvolatile memory register
Fermentation_001.MccRev_013.uMinutes       := FermentationProcess_001.fbDriveReverse_013.Minuts;           // PLC Work Time Counter - minutes nonvolatile memory register
Fermentation_001.MccRev_013.uSeconds       := FermentationProcess_001.fbDriveReverse_013.Seconds;          // PLC Work Time Counter - seconds nonvolatile memory register
Fermentation_001.MccRev_013.sState         := FermentationProcess_001.fbDriveReverse_013.MotorState;       // PLC Work Time Counter - minutes nonvolatile memory register
Fermentation_001.MccRev_013.sStatus        := FermentationProcess_001.fbDriveReverse_013.MotorStatus;      // PLC Work Time Counter - seconds nonvolatile memory register


//MccRev_014 variable sets by PLC
FermentationProcess_001.fbDriveReverse_014.MotorProtection := Fermentation_001.MccRev_014.bTermFuse;       // PLC input thermal fuse
Fermentation_001.MccRev_014.bContactor     := FermentationProcess_001.fbDriveReverse_014.MotorContactor;   // PLC output contactor
Fermentation_001.MccRev_014.udHours        := FermentationProcess_001.fbDriveReverse_014.Hours;            // PLC Work Time Counter - hours nonvolatile memory register
Fermentation_001.MccRev_014.uMinutes       := FermentationProcess_001.fbDriveReverse_014.Minuts;           // PLC Work Time Counter - minutes nonvolatile memory register
Fermentation_001.MccRev_014.uSeconds       := FermentationProcess_001.fbDriveReverse_014.Seconds;          // PLC Work Time Counter - seconds nonvolatile memory register
Fermentation_001.MccRev_014.sState         := FermentationProcess_001.fbDriveReverse_014.MotorState;       // PLC Work Time Counter - minutes nonvolatile memory register
Fermentation_001.MccRev_014.sStatus        := FermentationProcess_001.fbDriveReverse_014.MotorStatus;      // PLC Work Time Counter - seconds nonvolatile memory register

//MccRev_015 variable sets by PLC
FermentationProcess_001.fbDriveReverse_015.MotorProtection := Fermentation_001.MccRev_015.bTermFuse;       // PLC input thermal fuse
Fermentation_001.MccRev_015.bContactor     := FermentationProcess_001.fbDriveReverse_015.MotorContactor;   // PLC output contactor
Fermentation_001.MccRev_015.udHours        := FermentationProcess_001.fbDriveReverse_015.Hours;            // PLC Work Time Counter - hours nonvolatile memory register
Fermentation_001.MccRev_015.uMinutes       := FermentationProcess_001.fbDriveReverse_015.Minuts;           // PLC Work Time Counter - minutes nonvolatile memory register
Fermentation_001.MccRev_015.uSeconds       := FermentationProcess_001.fbDriveReverse_015.Seconds;          // PLC Work Time Counter - seconds nonvolatile memory register
Fermentation_001.MccRev_015.sState         := FermentationProcess_001.fbDriveReverse_015.MotorState;       // PLC Work Time Counter - minutes nonvolatile memory register
Fermentation_001.MccRev_015.sStatus        := FermentationProcess_001.fbDriveReverse_015.MotorStatus;      // PLC Work Time Counter - seconds nonvolatile memory register


//MccRev_016 variable sets by PLC
FermentationProcess_001.fbDriveReverse_016.MotorProtection := Fermentation_001.MccRev_016.bTermFuse;       // PLC input thermal fuse
Fermentation_001.MccRev_016.bContactor     := FermentationProcess_001.fbDriveReverse_016.MotorContactor;   // PLC output contactor
Fermentation_001.MccRev_016.udHours        := FermentationProcess_001.fbDriveReverse_016.Hours;            // PLC Work Time Counter - hours nonvolatile memory register
Fermentation_001.MccRev_016.uMinutes       := FermentationProcess_001.fbDriveReverse_016.Minuts;           // PLC Work Time Counter - minutes nonvolatile memory register
Fermentation_001.MccRev_016.uSeconds       := FermentationProcess_001.fbDriveReverse_016.Seconds;          // PLC Work Time Counter - seconds nonvolatile memory register
Fermentation_001.MccRev_016.sState         := FermentationProcess_001.fbDriveReverse_016.MotorState;       // PLC Work Time Counter - minutes nonvolatile memory register
Fermentation_001.MccRev_016.sStatus        := FermentationProcess_001.fbDriveReverse_016.MotorStatus;      // PLC Work Time Counter - seconds nonvolatile memory register


//MccRev_017 variable sets by PLC
FermentationProcess_001.fbDriveReverse_017.MotorProtection := Fermentation_001.MccRev_017.bTermFuse;       // PLC input thermal fuse
Fermentation_001.MccRev_017.bContactor     := FermentationProcess_001.fbDriveReverse_017.MotorContactor;   // PLC output contactor
Fermentation_001.MccRev_017.udHours        := FermentationProcess_001.fbDriveReverse_017.Hours;            // PLC Work Time Counter - hours nonvolatile memory register
Fermentation_001.MccRev_017.uMinutes       := FermentationProcess_001.fbDriveReverse_017.Minuts;           // PLC Work Time Counter - minutes nonvolatile memory register
Fermentation_001.MccRev_017.uSeconds       := FermentationProcess_001.fbDriveReverse_017.Seconds;          // PLC Work Time Counter - seconds nonvolatile memory register
Fermentation_001.MccRev_017.sState         := FermentationProcess_001.fbDriveReverse_017.MotorState;       // PLC Work Time Counter - minutes nonvolatile memory register
Fermentation_001.MccRev_017.sStatus        := FermentationProcess_001.fbDriveReverse_017.MotorStatus;      // PLC Work Time Counter - seconds nonvolatile memory register


//MccRev_018 variable sets by PLC
FermentationProcess_001.fbDriveReverse_018.MotorProtection := Fermentation_001.MccRev_018.bTermFuse;       // PLC input thermal fuse
Fermentation_001.MccRev_018.bContactor     := FermentationProcess_001.fbDriveReverse_018.MotorContactor;   // PLC output contactor
Fermentation_001.MccRev_018.udHours        := FermentationProcess_001.fbDriveReverse_018.Hours;            // PLC Work Time Counter - hours nonvolatile memory register
Fermentation_001.MccRev_018.uMinutes       := FermentationProcess_001.fbDriveReverse_018.Minuts;           // PLC Work Time Counter - minutes nonvolatile memory register
Fermentation_001.MccRev_018.uSeconds       := FermentationProcess_001.fbDriveReverse_018.Seconds;          // PLC Work Time Counter - seconds nonvolatile memory register
Fermentation_001.MccRev_018.sState         := FermentationProcess_001.fbDriveReverse_018.MotorState;       // PLC Work Time Counter - minutes nonvolatile memory register
Fermentation_001.MccRev_018.sStatus        := FermentationProcess_001.fbDriveReverse_018.MotorStatus;      // PLC Work Time Counter - seconds nonvolatile memory register


//MccRev_019 variable sets by PLC
FermentationProcess_001.fbDriveReverse_019.MotorProtection := Fermentation_001.MccRev_019.bTermFuse;       // PLC input thermal fuse
Fermentation_001.MccRev_019.bContactor     := FermentationProcess_001.fbDriveReverse_019.MotorContactor;   // PLC output contactor
Fermentation_001.MccRev_019.udHours        := FermentationProcess_001.fbDriveReverse_019.Hours;            // PLC Work Time Counter - hours nonvolatile memory register
Fermentation_001.MccRev_019.uMinutes       := FermentationProcess_001.fbDriveReverse_019.Minuts;           // PLC Work Time Counter - minutes nonvolatile memory register
Fermentation_001.MccRev_019.uSeconds       := FermentationProcess_001.fbDriveReverse_019.Seconds;          // PLC Work Time Counter - seconds nonvolatile memory register
Fermentation_001.MccRev_019.sState         := FermentationProcess_001.fbDriveReverse_019.MotorState;       // PLC Work Time Counter - minutes nonvolatile memory register
Fermentation_001.MccRev_019.sStatus        := FermentationProcess_001.fbDriveReverse_019.MotorStatus;      // PLC Work Time Counter - seconds nonvolatile memory register


//MccRev_020 variable sets by PLC
FermentationProcess_001.fbDriveReverse_020.MotorProtection := Fermentation_001.MccRev_020.bTermFuse;       // PLC input thermal fuse
Fermentation_001.MccRev_020.bContactor     := FermentationProcess_001.fbDriveReverse_020.MotorContactor;   // PLC output contactor
Fermentation_001.MccRev_020.udHours        := FermentationProcess_001.fbDriveReverse_020.Hours;            // PLC Work Time Counter - hours nonvolatile memory register
Fermentation_001.MccRev_020.uMinutes       := FermentationProcess_001.fbDriveReverse_020.Minuts;           // PLC Work Time Counter - minutes nonvolatile memory register
Fermentation_001.MccRev_020.uSeconds       := FermentationProcess_001.fbDriveReverse_020.Seconds;          // PLC Work Time Counter - seconds nonvolatile memory register
Fermentation_001.MccRev_020.sState         := FermentationProcess_001.fbDriveReverse_020.MotorState;       // PLC Work Time Counter - minutes nonvolatile memory register
Fermentation_001.MccRev_020.sStatus        := FermentationProcess_001.fbDriveReverse_020.MotorStatus;      // PLC Work Time Counter - seconds nonvolatile memory register
END_ACTION

ACTION ACT_PhSens:
fbPhSens_001(
    _rX := Fermentation_001.PhSens_001.rRawPhValue,
    _rXmin := 0,
    _rXmax := 32767,
    _rYmin := 0,
    _rYmax := 12); // FB_Scaling
Fermentation_001.PhSens_001.rPhValue := fbPhSens_001._rY;
END_ACTION

ACTION ACT_PressureSens:
fbPressureSens_001(
    _rX := Fermentation_001.PhSens_001.rRawPhValue,
    _rXmin := 0,
    _rXmax := 32767,
    _rYmin := 0,
    _rYmax := 12); // FB_Scaling
Fermentation_001.PhSens_001.rPhValue := fbPressureSens_001._rY;
END_ACTION

ACTION ACT_TempSens:
fbTempSens_003(
    _rX := Fermentation_001.TempSens_003.rRawTempValue,
    _rXmin := 0,
    _rXmax := 32767,
    _rYmin := 0,
    _rYmax := 100); // FB_Scaling
fbTempSens_001(
    _rX := Fermentation_001.TempSens_001.rRawTempValue,
    _rXmin := 0,
    _rXmax := 32767,
    _rYmin := 0,
    _rYmax := 100); // FB_Scaling
Fermentation_001.TempSens_003.rTempValue := fbTempSens_003._rY;
Fermentation_001.TempSens_001.rTempValue := fbTempSens_001._rY;
fbTempSens_002(
    _rX := Fermentation_001.TempSens_002.rRawTempValue,
    _rXmin := 0,
    _rXmax := 32767,
    _rYmin := 0,
    _rYmax := 100); // FB_Scaling
Fermentation_001.TempSens_002.rTempValue := fbTempSens_002._rY;
END_ACTION

END_PROGRAM

// ---- POUs/Implementation/FB_DriveReverse.TcPOU
FUNCTION_BLOCK FB_DriveReverse EXTENDS FB_Drive IMPLEMENTS I_DriveReverse

VAR
	_contactorReverse		: ContactorReverse;	// załącz/wyłącz stycznik do tyłu silnika

END_VAR

METHOD StatusState : E_StateDevice
VAR_INPUT
END_VAR
// State Machine of the Drive 
// zliczaj czas pracy gdy napęd jest uruchomiony




CASE _eStateMachine OF
	
	eOff:
		WorkCounterOff();
		_supplyLed.State := FALSE;
		_stateLabel.Text := 'OFF';
		_statusLabel.Text := 'Napęd jest wyłączony';
		_contactor.State := FALSE;
		_contactorReverse.State := FALSE;
		
		IF (_eCommand = eReady) AND _termFuse.IsActive THEN
			_eStateMachine := eOn;	
		END_IF
	
	eOn:
		WorkCounterOff();
		_supplyLed.State := TRUE;
		_stateLabel.Text := 'ON';
		_statusLabel.Text := 'Napęd jest w gotowości';
		_contactor.State := FALSE;
		_contactorReverse.State := FALSE;

		IF _eCommand = eFwd THEN
			_eStateMachine := eForward;
		ELSIF _eCommand = eRev THEN
			_eStateMachine := eReverse;
		ELSIF _eCommand = eReady AND NOT _termFuse.IsActive THEN
			_eStateMachine := eOff;
		ELSIF _eCommand = eReady AND _termFuse.IsActive THEN
			_eStateMachine := eOn;	
		END_IF
		
	
	eForward:
		_stateLabel.Text := 'RUNNING';
		_statusLabel.Text := 'Napęd jest uruchomiony do przodu';	
		WorkCounterOn();
		WorkCount();
		WorkTimelabel();	
		IF _eCommand = eFwd THEN
			_contactor.State := TRUE;
		ELSIF _eCommand = eReady THEN
			_eStateMachine := eOn;
		END_IF
		
        IF _eCommand = eFwd AND NOT _termFuse.IsActive THEN
			_eStateMachine := eFault;
		END_IF
		
	eReverse:
		_stateLabel.Text := 'RUNNING';
		_statusLabel.Text := 'Napęd jest uruchomiony do tyłu';	
		WorkCounterOn();
		WorkCount();
		WorkTimelabel();
		IF _eCommand = eRev THEN
			_contactorReverse.State := TRUE;
		ELSIF _eCommand = eReady THEN
			_eStateMachine := eOn;
		END_IF
		
        IF _eCommand = eRev AND NOT _termFuse.IsActive THEN
			_eStateMachine := eFault;
		END_IF		
	
		
	eFault:
		_contactor.State := FALSE;
		_contactorReverse.State := FALSE;
		WorkCounterOff();
		_stateLabel.Text := 'FAULT';
		_statusLabel.Text := 'Zadziałał wyłacznik silnikowy';
		IF _eCommand = eReady AND NOT _termFuse.IsActive THEN
			_eStateMachine := eOff;
		END_IF

END_CASE




//IF _termFuse.IsActive THEN
//		_supplyLed.State := TRUE;
//		_stateLabel.Text := 'ON';
//		_statusLabel.Text := 'Napęd jest w gotowości';	
//		StatusState := eOn;

//	IF _contactor.State THEN
//		_stateLabel.Text := 'RUNNING';
//		_statusLabel.Text := 'Napęd jest uruchomiony do przodu';
		
//		// start count work time
//		WorkTimelabel();
//		StatusState := eForward;
//	END_IF
	
//	IF _contactorReverse.State THEN
//		_stateLabel.Text := 'RUNNING';
//		_statusLabel.Text := 'Napęd jest uruchomiony do tyłu';
		
//		// start count work time
//		WorkTimelabel();
//		StatusState := eReverse;
//	END_IF
	
	
//ELSE
//		_supplyLed.State := FALSE;
//		_stateLabel.Text := 'OFF';
//		_statusLabel.Text := 'Napęd jest wyłączony';
//		StatusState := eOff;

//	IF _contactor.State OR _contactorReverse.State THEN
//		_stateLabel.Text := 'FAULT';
//		_statusLabel.Text := 'Zadziałał wyłacznik silnikowy';
//		StatusState := eFault;
//	END_IF

//END_IF
END_METHOD

METHOD SwitchReverseOff : BOOL
THIS^._eCommand := eReady;
END_METHOD

METHOD SwitchReverseOn : BOOL
THIS^._eCommand := eRev;
END_METHOD

END_FUNCTION_BLOCK

// ---- POUs/Implementation/FB_Drive.TcPOU
FUNCTION_BLOCK FB_Drive IMPLEMENTS I_Drive
VAR
	//_test			: -(GVL.bAuto);
	_contactor		: Contactor;	// załącz/wyłącz stycznik silnika
	_autoLed 		: Led;	// zaświeć/zgaś Led auto w stacyjce napędu SCADA
	_supplyLed		: Led;	// zaświeć/zgaś Led supply w stacyjce napędu SCADA
	_stateLabel		: Label; // label do wyświetlania stanu urzadzenia w stacyjce SCADA
	_workTimeLabel	: Label; // label do wyświetlania czasu pracy napędu w stacyjce SCADA
	_statusLabel	: Label; // label to wyświetlania statusu napędu w stacyjce SCADA
	_termFuse		: TermFuse; // wejście zabezpieczenia termicznego i nadprądowego napędu
	_text			: T_MaxString;

	_startCount  	: BOOL;		// start/stop zliczania czasu
	_stWorkTime  	: ST_WorkTime;	// struktura czasu pracy napędu

	_eStateMachine	: E_StateDevice :=eOff; //Drive State Machine ustaw stan początkowy
	_eCommand		: E_Command;     // Command
  
END_VAR

METHOD AutoLedOff : BOOL
VAR_INPUT
END_VAR
_autoLed.State := FALSE;
END_METHOD

METHOD AutoLedOn : BOOL
VAR_INPUT
END_VAR
_autoLed.State := TRUE;
END_METHOD

PROPERTY Hours : UDINT
GET
Hours := _stWorkTime.hours;
END_GET
SET
_stWorkTime.hours := Hours;
END_SET
END_PROPERTY

PROPERTY Minuts : UINT
GET
Minuts := _stWorkTime.minuts;
END_GET
SET
_stWorkTime.minuts := Minuts;
END_SET
END_PROPERTY

PROPERTY MotorAuto : BOOL
GET
MotorAuto := _autoLed.State;
END_GET
SET
_autoLed.State := MotorAuto;
END_SET
END_PROPERTY

PROPERTY MotorContactor : BOOL
GET
MotorContactor := _contactor.State;
END_GET
SET
_contactor.State := MotorContactor;
END_SET
END_PROPERTY

PROPERTY MotorProtection : BOOL
GET
MotorProtection := _termFuse.IsActive;
END_GET
SET
_termFuse.IsActive := MotorProtection;
END_SET
END_PROPERTY

PROPERTY MotorState : T_MaxString
GET
MotorState := _stateLabel.Text;
END_GET
SET
_stateLabel.Text := MotorState;
END_SET
END_PROPERTY

PROPERTY MotorStatus : T_MaxString
GET
MotorStatus := _statusLabel.Text;
END_GET
SET
_statusLabel.Text := MotorStatus;
END_SET
END_PROPERTY

PROPERTY MotorSupply : BOOL
GET
MotorSupply := _supplyLed.State;
END_GET
END_PROPERTY

PROPERTY Seconds : UINT
GET
Seconds := _stWorkTime.seconds;
END_GET
SET
_stWorkTime.seconds := Seconds;
END_SET
END_PROPERTY

METHOD StatusState : E_StateDevice
VAR_INPUT
END_VAR
// State Machine of the Drive 
// zliczaj czas pracy gdy napęd jest uruchomiony


CASE _eStateMachine OF
	
	eOff:
		WorkCounterOff();
		_supplyLed.State := FALSE;
		_stateLabel.Text := 'OFF';
		_statusLabel.Text := 'Napęd jest wyłączony';
		_contactor.State := FALSE;
		
		IF (_eCommand = eReady) AND _termFuse.IsActive THEN
			_eStateMachine := eOn;	
		END_IF
	
	eOn:
		WorkCounterOff();
		_supplyLed.State := TRUE;
		_stateLabel.Text := 'ON';
		_statusLabel.Text := 'Napęd jest w gotowości';
		_contactor.State := FALSE;

		IF _eCommand = eFwd THEN
			_eStateMachine := eForward;
		ELSIF _eCommand = eReady AND NOT _termFuse.IsActive THEN
			_eStateMachine := eOff;
		ELSIF _eCommand = eReady AND _termFuse.IsActive THEN
			_eStateMachine := eOn;	
		END_IF
		
	
	eForward:
		_stateLabel.Text := 'RUNNING';
		_statusLabel.Text := 'Napęd jest uruchomiony do przodu';	
		WorkCounterOn();
		WorkCount();
		WorkTimelabel();	
		IF _eCommand = eFwd THEN
			_contactor.State := TRUE;
		ELSIF _eCommand = eReady THEN
			_eStateMachine := eOn;
		END_IF
		
        IF _eCommand = eFwd AND NOT _termFuse.IsActive THEN
			_eStateMachine := eFault;
		END_IF
		
	
	eFault:
		_contactor.State := FALSE;
		WorkCounterOff();
		_stateLabel.Text := 'FAULT';
		_statusLabel.Text := 'Zadziałał wyłacznik silnikowy';
		IF _eCommand = eReady AND NOT _termFuse.IsActive THEN
			_eStateMachine := eOff;
		END_IF

END_CASE





//IF _termFuse.IsActive THEN
//		_supplyLed.State := TRUE;
//		_stateLabel.Text := 'ON';
//		_statusLabel.Text := 'Napęd jest w gotowości';
//		StatusState := eOn;
		
//	IF _contactor.State THEN
//		_stateLabel.Text := 'RUNNING';
//		_statusLabel.Text := 'Napęd jest uruchomiony do przodu';
		
//		// start count work time
//		WorkTimelabel();
//		StatusState := eForward;
		
		
//	END_IF

//ELSE
//		_supplyLed.State := FALSE;
//		_stateLabel.Text := 'OFF';
//		_statusLabel.Text := 'Napęd jest wyłączony';
//		StatusState := eOff;

//	IF _contactor.State THEN
//		_stateLabel.Text := 'FAULT';
//		_statusLabel.Text := 'Zadziałał wyłacznik silnikowy';
//		StatusState := eFault;
//	END_IF

//END_IF
END_METHOD

METHOD SwitchOff : BOOL
VAR_INPUT
	
END_VAR
_eCommand := eReady;
END_METHOD

METHOD SwitchOn : BOOL
VAR_INPUT
END_VAR
_eCommand := eFwd;
END_METHOD

METHOD PUBLIC WorkCount : STRING
VAR_INPUT
END_VAR

VAR_INST
	fbTon	: TON;
END_VAR
fbTon(IN := _startCount, PT := T#1S);

IF (fbTon.Q) THEN
	
	fbTon(IN:=FALSE);
	_stWorkTime.seconds := _stWorkTime.seconds +1;
	
	IF _stWorkTime.seconds > 59 THEN
		_stWorkTime.seconds := 0;
		_stWorkTime.minuts := _stWorkTime.minuts +1;
		IF _stWorkTime.minuts > 59 THEN
			_stWorkTime.minuts := 0;
			_stWorkTime.hours := _stWorkTime.hours +1;	
		END_IF
	END_IF
	
END_IF
END_METHOD

METHOD WorkCounterOff : BOOL
VAR_INPUT
END_VAR
_startCount := FALSE;
END_METHOD

METHOD WorkCounterOn : BOOL
VAR_INPUT
END_VAR
_startCount := TRUE;
END_METHOD

METHOD PROTECTED WorkTimeLabel : STRING
VAR_INPUT
END_VAR
// Forms a chain of the form 'Hours:Minuts:Seconds'
_text := CONCAT(UDINT_TO_STRING(THIS^._stWorkTime.hours), ':');
_text := CONCAT(_text, UDINT_TO_STRING(THIS^._stWorkTime.minuts));
_text := CONCAT(_text, ':');
_text := CONCAT(_text, UDINT_TO_STRING(_stWorkTime.seconds));

_workTimeLabel.Text := _text;
END_METHOD

END_FUNCTION_BLOCK

// ---- POUs/Devices/Contactor.TcPOU
FUNCTION_BLOCK Contactor
VAR
	_output : BOOL;
END_VAR

PROPERTY State : BOOL
GET
State := _output;
END_GET
SET
_output := State;
END_SET
END_PROPERTY

END_FUNCTION_BLOCK

// ---- POUs/Devices/Led.TcPOU
FUNCTION_BLOCK Led
VAR
	_state : BOOL;
END_VAR

PROPERTY State : BOOL
GET
State := _state;
END_GET
SET
_state := State;
END_SET
END_PROPERTY

END_FUNCTION_BLOCK

// ---- POUs/Devices/Label.TcPOU
FUNCTION_BLOCK Label 
VAR
	_label : T_MaxString;
END_VAR

PROPERTY Text : STRING
GET
Text := _label;
END_GET
SET
_label := Text;
END_SET
END_PROPERTY

END_FUNCTION_BLOCK

// ---- POUs/Devices/TermFuse.TcPOU
FUNCTION_BLOCK TermFuse
VAR
	_input : BOOL;
	
END_VAR

PROPERTY IsActive : BOOL
GET
IsActive := _input;
END_GET
SET
_input := IsActive;
END_SET
END_PROPERTY

END_FUNCTION_BLOCK

// ---- POUs/Devices/ContactorReverse.TcPOU
FUNCTION_BLOCK ContactorReverse
VAR
	_output  : BOOL;
END_VAR

PROPERTY State : BOOL
GET
State := _output;
END_GET
SET
_output := State;
END_SET
END_PROPERTY

END_FUNCTION_BLOCK

// ---- POUs/Abstraction/FB_MotorControlReverse.TcPOU
FUNCTION_BLOCK FB_MotorControlReverse EXTENDS FB_MotorControl
VAR
	reverseButton		: Button;	// Scada Button reverse
	iDriveReverse		: I_DriveReverse; //Interface variable 
	
	bSuccess: BOOL;
	
END_VAR

SUPER^(); //call base class 



//Button Auto is set in SCADA motor control station, but Client in PLC have to have acces too directly via a variable to work in Auto mode
IF autoButton.IsPressed THEN 
	AutoOn();	// Turn On SCADA auto Led

ELSE
	AutoOff(); // Turn Off SCADA auto Led
	
	// IF NOT AUTO MODE THEN, EXECUTE
	
	IF reverseButton.IsPressed THEN
		ReverseOn();
	ELSIF NOT forwardButton.IsPressed THEN
		ReverseOff();
	END_IF

END_IF

METHOD FB_init : BOOL
VAR_INPUT
	bInitRetains : BOOL; // if TRUE, the retain variables are initialized (warm start / cold start)
	bInCopyCode  : BOOL;  // if TRUE, the instance afterwards gets moved into the copy code (online change)
	iDrive		 : I_Drive;
			
END_VAR
//check it is possible conversion type of interface

IF __QUERYINTERFACE(iDrive, iDriveReverse) THEN
	bSuccess := TRUE;
END_IF
END_METHOD

METHOD ReverseOff : BOOL
VAR_INPUT
END_VAR
ReverseOff := iDriveReverse.SwitchReverseOff();
END_METHOD

METHOD ReverseOn : BOOL
VAR_INPUT
END_VAR
ReverseOn := iDriveReverse.SwitchReverseOn();
END_METHOD

PROPERTY ScadaReverseButton : BOOL
GET
ScadaReverseButton := reverseButton.IsPressed;
END_GET
SET
reverseButton.IsPressed := ScadaReverseButton;
END_SET
END_PROPERTY

END_FUNCTION_BLOCK

// ---- POUs/Abstraction/FB_MotorControl.TcPOU
// Function block to control simple MCC 
FUNCTION_BLOCK FB_MotorControl
VAR
	autoButton		    : Button;	   // Scada Button auto
	forwardButton	    : Button;	   // Scada Button forward
	iDrive 		        : I_Drive;     // interface variable
		
END_VAR

// Run State Machine of The Drive
iDrive.StatusState();



//Button Auto is set in SCADA motor control station, but Client in PLC have to have acces too directly via a variable to work in Auto mode
IF autoButton.IsPressed THEN 
	AutoOn();	// Turn On SCADA auto Led

ELSE
	AutoOff(); // Turn Off SCADA auto Led
	
	// IF NOT AUTO MODE THEN, EXECUTE

	
	IF forwardButton.IsPressed THEN
		ForwardOn();
	ELSE
		ForwardOff();
	END_IF
	

END_IF

METHOD PUBLIC AutoOff : BOOL
VAR_INPUT
END_VAR
iDrive.AutoLedOff();
END_METHOD

METHOD PUBLIC AutoOn : BOOL
VAR_INPUT
END_VAR
iDrive.AutoLedOn();
END_METHOD

METHOD FB_init : BOOL
VAR_INPUT
	bInitRetains : BOOL; // if TRUE, the retain variables are initialized (warm start / cold start)
	bInCopyCode  : BOOL;  // if TRUE, the instance afterwards gets moved into the copy code (online change)
	iDrive		 : I_Drive;
END_VAR
THIS^.iDrive := iDrive;
END_METHOD

METHOD PUBLIC ForwardOff : BOOL
VAR_INPUT

END_VAR
ForwardOff := iDrive.SwitchOff();
END_METHOD

METHOD PUBLIC ForwardOn : BOOL
VAR_INPUT

END_VAR
ForwardOn := iDrive.SwitchOn();
END_METHOD

PROPERTY ScadaAutoButton : BOOL
GET
ScadaAutoButton := autoButton.IsPressed;
END_GET
SET
autoButton.IsPressed :=  ScadaAutoButton;
END_SET
END_PROPERTY

PROPERTY ScadaForwardButton : BOOL
GET
ScadaForwardButton := forwardButton.IsPressed;
END_GET
SET
forwardButton.IsPressed := ScadaForwardButton;
END_SET
END_PROPERTY

END_FUNCTION_BLOCK

// ---- POUs/Devices/Button.TcPOU
FUNCTION_BLOCK Button
VAR
	_input	: BOOL;
END_VAR

PROPERTY IsPressed : BOOL
GET
IsPressed:= _input;
END_GET
SET
_input := IsPressed;
END_SET
END_PROPERTY

END_FUNCTION_BLOCK

// ---- POUs/Scaling/FB_Scaling.TcPOU
FUNCTION_BLOCK FB_Scaling
VAR
	_rA		: REAL;		// factor 'a' in linear equation
	_rB		: REAL;		// factor 'b' in linear equation	 
END_VAR

VAR_INPUT
	_rX     : REAL; 	// input value
	_rXmin  : REAL;		// low value of input range
	_rXmax  : REAL;		// high value of input range
	_rYmin  : REAL;		// low value of output range
	_rYmax  : REAL;		// high value of output range
END_VAR

VAR_OUTPUT
	_bAlarmHi: BOOL;
	_bAlarmLo: BOOL;
	_rY: REAL;
END_VAR

IF ABS (_rXmax - _rXmin) > 0.01 THEN 
	IF _rX <= _rXmin THEN 
		_bAlarmLo := TRUE; 
        _bAlarmHi := FALSE; 
		_rY := _rYmin; 
	ELSIF _rX >= _rXmax THEN 
		_bAlarmLo := FALSE; 
		_bAlarmHi := TRUE; 
		_rY := _rYmax; 
	ELSE 
		_bAlarmLo := FALSE; 
		_bAlarmHi := FALSE; 
		_rA := (_rYmax - _rYmin)/(_rXmax - _rXmin); 
		_rB := _rYmax - _rA *_rXmax; 
		_rY := _rA * _rX + _rB; 
	END_IF 
ELSE 
	_rY := _rYmin; 
	_bAlarmHi := TRUE; 
	_bAlarmLo := TRUE;
END_IF

END_FUNCTION_BLOCK

// ---- POUs/Abstraction/FB_MotorControlInverter.TcPOU
FUNCTION_BLOCK FB_MotorControlInverter EXTENDS FB_MotorControlReverse
VAR
	resetButton		: Button;	   // Scada Button inverter reset
	speedEdit		: NumberEdit; // SCADA number Edit field
	
	iDriveInverter  : I_DriveInverter; // interface variable
	
	
END_VAR

SUPER^(); //call base class 


//Button Auto is set in SCADA motor control station, but Client in PLC have to have acces too directly via a variable to work in Auto mode
IF autoButton.IsPressed THEN 
	AutoOn();	// Turn On SCADA auto Led
ELSE
	AutoOff(); // Turn Off SCADA auto Led
	
	// IF NOT AUTO MODE THEN, EXECUTE
	
	 IF resetButton.IsPressed THEN
		Reset();		
	 END_IF
				 

END_IF


// Speed set all the time
Speed(speedEdit.Number);

METHOD FB_init : BOOL
VAR_INPUT
	bInitRetains : BOOL; // if TRUE, the retain variables are initialized (warm start / cold start)
	bInCopyCode  : BOOL;  // if TRUE, the instance afterwards gets moved into the copy code (online change)
	iDrive		 : I_Drive;
			
END_VAR
//check it is possible conversion type of interface

IF __QUERYINTERFACE(iDrive, iDriveInverter) THEN
	bSuccess := TRUE;
END_IF
END_METHOD

METHOD Reset : BOOL
VAR_INPUT
END_VAR
iDriveInverter.Reset();
END_METHOD

PROPERTY ScadaResetButton : BOOL
GET
ScadaResetButton := resetButton.IsPressed;
END_GET
END_PROPERTY

PROPERTY ScadaSpeedEdit : REAL
GET
ScadaSpeedEdit := speedEdit.Number;
END_GET
END_PROPERTY

METHOD Speed : BOOL
VAR_INPUT
	_setSpeedValue : REAL;
END_VAR
iDriveInverter.SetSpeed(_setSpeedValue);
END_METHOD

END_FUNCTION_BLOCK

// ---- POUs/Devices/NumberEdit.TcPOU
FUNCTION_BLOCK NumberEdit
VAR
	_number : REAL;
END_VAR

PROPERTY Number : REAL
GET
Number := _number;
END_GET
SET
_number := Number;
END_SET
END_PROPERTY

END_FUNCTION_BLOCK

// ---- POUs/Devices/Button_1.TcPOU
FUNCTION_BLOCK Button_1
VAR
	_input	: REFERENCE TO BOOL;
END_VAR

METHOD FB_init : BOOL
VAR_INPUT
	bInitRetains : BOOL; // if TRUE, the retain variables are initialized (warm start / cold start)
	bInCopyCode : BOOL;  // if TRUE, the instance afterwards gets moved into the copy code (online change)
	_input : REFERENCE TO BOOL;
END_VAR
THIS^._input REF= _input;
END_METHOD

PROPERTY IsPressed : BOOL
GET
IsPressed:= _input;
END_GET
END_PROPERTY

END_FUNCTION_BLOCK

// ---- POUs/Devices/Modbus/FB_InverterOperation.TcPOU
FUNCTION_BLOCK FB_InverterOperation

VAR
	
	MB           		: ModbusRtuMaster_KL6x22B;
	_MBdata      		: ARRAY[0..40] OF WORD;	(* The size of this array can be adapted to the modbus slaves register area *)
 	_busy		 		: BOOL;	
	_timeoutvalue		: TIME:=T#300MS;		            (* Timeout while waiting for an answer of the modbus slave *)
	
	_step		 		: INT;						(* Step of the control inverter program*)
	_iItfCount			: INT :=1;
	_stInverter			: ST_Inverter;
	


	
	

END_VAR

CASE _step OF
0:	(*Initialize*)
		MB.ReadRegs(Execute:= FALSE); (* initialize *)
		
		//set index of inverter FB  
		_iItfCount := 1;		
		_step:= 10;

10:	(*Read status of Inverter*) (*Sprawdzić status po wystąpieniu bledu przerwania komuikacji*)

		// Read the device settings
		_stInverter := Itf.aItfDriveInverter[_iItfCount].DeviceData;
		
		MB.ReadRegs(
			UnitID:=_stInverter.bDeviceId,
			Quantity:= 1,
			MBAddr:=3201,
			cbLength:= 2,
			pMemoryAddr:= ADR(_MBdata[0]),
			Execute:= TRUE,
			Timeout:= _timeoutvalue,
			Busy => _busy	);


		IF NOT _busy THEN	
			MB.ReadRegs(Execute:=FALSE);
			_stInverter.errorMdb := MB.ErrorId;		
		
			IF NOT MB.Error THEN
				_stInverter.wStatus := StatusWord(_MBdata);
				_step :=20;
			END_IF		
			
		END_IF


	
		
20: 	(*Write Control Register*)

		CASE _stInverter.eControl OF
			eShutDown:
				_MBdata[0] := eShutDown;			
			eSwitchOn:
				_MBdata[0] := eSwitchOn;
			eEnableOperation:
			   _MBdata[0] := eEnableOperation;
			eReverseOperation:
				_MBdata[0] := eReverseOperation;
			eFaultReset:
				_MBdata[0] := eFaultReset;
						 
		ELSE
			_MBdata[0] := 0;
		
		END_CASE	

			
		MB.WriteSingleRegister(
			UnitID:=_stInverter.bDeviceId,
			Quantity:=1,
			MBAddr:=8501,
			cbLength:= 2,
			pMemoryAddr:= ADR(_MBdata[0]),
			Execute:= TRUE,
			Timeout:= _timeoutvalue,
			Busy => _busy	);

		IF NOT _busy THEN
			MB.ReadRegs(Execute:=FALSE);
			_step := 30;
		END_IF

30: 	(*Write the set frequency*)
		
		_MBdata[0] := _stInverter.rSpeed;
	
		MB.WriteSingleRegister(
					UnitID:=_stInverter.bDeviceId,
					Quantity:=1,
					MBAddr:=8502,
					cbLength:= 2,
					pMemoryAddr:= ADR(_MBdata[0]),
					Execute:= TRUE,
					Timeout:= _timeoutvalue,
					Busy => _busy	);
	
		IF NOT _busy THEN
			MB.WriteRegs(Execute:=FALSE);
			_step :=40;
		END_IF
		

40:	(*Read actual error of Inverter*)
	
		MB.ReadRegs(
			UnitID:=_stInverter.bDeviceId,
			Quantity:= 1,
			MBAddr:=7200,
			cbLength:= 2,
			pMemoryAddr:= ADR(_MBdata[0]),
			Execute:= TRUE,
			Timeout:= _timeoutvalue,
			Busy => _busy	);
			
		IF NOT _busy THEN
			MB.ReadRegs(Execute:=FALSE);
			_stInverter.errorMdb := MB.ErrorId;			
			IF NOT MB.Error THEN
				_stInverter.errorInv := ErrorWord(_MBdata, sErrorDescription => _stInverter.sErrorDescription);
			END_IF
	
			_MBdata[0]:=0;
			_step :=50;	
			
			Itf.aItfDriveInverter[_iItfCount].DeviceData := _stInverter;	
		END_IF
		
50: (* Go to the next device*)
	
	IF _iItfCount < Itf.aItfDriveInverter[_iItfCount].InstanceCounter THEN
		_iItfCount := _iItfCount +1;
		_step := 10;
	ELSE
		_step := 0;
		
	END_IF


	
END_CASE

METHOD ErrorWord : E_InverterError
VAR_INPUT
	refMBdata : REFERENCE TO ARRAY[0..40] OF WORD;  //wskaźnik do tablicy ze słowem błędu Error Inverter
END_VAR


VAR_OUTPUT
	
	sErrorDescription : T_MaxString;
END_VAR


CASE refMBdata[0] OF
	
	0:
		ErrorWord := 0;
		sErrorDescription := 'Brak Błędu';
	1: 
		ErrorWord := 1;
		sErrorDescription := 'Błąd InF';
	3: 
		ErrorWord := 3;
		sErrorDescription := 'Incorrect Configuration';
	4:
		ErrorWord := 4;
		sErrorDescription := 'Incvalid Configuration'; 
	5:
		ErrorWord := 5;
		sErrorDescription := 'Modbus communications - interruption in communication on the Modbus network' ;
	8:
		ErrorWord := 8;
		sErrorDescription := 'External detected fault by logic input'; 
	9: 
		ErrorWord := 9;
		sErrorDescription := 'Overcurrent';
	10: 
		ErrorWord := 10;
		sErrorDescription := 'Precharge - Charging relay control fault or charging resistor damaged';
	16:
		ErrorWord := 16;
		sErrorDescription := 'Overheat - Drive temperature to high'; 
	17:
		ErrorWord := 17;
		sErrorDescription := 'Motor overload - triggered by excessive motor current'; 
	18:
		ErrorWord := 18;
		sErrorDescription :=  'Overbraking - Braking too sudden or driving load too high';
	19: 
		ErrorWord := 19;
		sErrorDescription := 'Main Overvoltage - line voltage to high';
	20: 
		ErrorWord := 20;
		sErrorDescription := '1 output phases loss';
	21:
		ErrorWord := 21;
		sErrorDescription := 'Input phase loss';
	22:
		ErrorWord := 22;
		sErrorDescription := 'Undervoltage';
	23:
		ErrorWord := 23;
		sErrorDescription := 'Motor or Ground short circuit';
	24: 
		ErrorWord := 24;
		sErrorDescription := 'Overspeed';
	25: 
		ErrorWord := 25;
		sErrorDescription := 'Auto-tunning';
	26:
		ErrorWord := 26;
		sErrorDescription := 'Unknown drive rating';
	27:
		ErrorWord := 27;
		sErrorDescription := 'Unknown or incompatible power board';
	28:
		ErrorWord := 28;
		sErrorDescription := 'Internal serial link'; 
	29:
		ErrorWord := 29;
		sErrorDescription := 'Invalid industrialization zone'; 
	32: 
		ErrorWord := 32;
		sErrorDescription :='Ground short circuit'; 
	33: 
		ErrorWord := 33;
		sErrorDescription := '3 output phase loss';
	42:
		ErrorWord := 42;
		sErrorDescription := 'SoMove communication - interruption';
	45:
		ErrorWord := 45;
		sErrorDescription := 'HMI communication - interruption';
	51:
		ErrorWord := 51;
		sErrorDescription := 'Current measurement circuit';
	53: 
		ErrorWord := 53;
		sErrorDescription := 'Internal thermal sensor detected fault'; 
	54: 
		ErrorWord := 54;
		sErrorDescription := 'IGBT overheat '; 
	55:
		ErrorWord := 55;
		sErrorDescription := 'IGBT short circuit'; 
	56:
		ErrorWord := 56;
		sErrorDescription := 'Load short circuit';
	69:
		ErrorWord := 69;
		sErrorDescription := 'Internal CPU'; 
	77: 
		ErrorWord := 77;
		sErrorDescription := 'Download invalid configuration'; 
	100: 
		ErrorWord := 100;
		sErrorDescription := 'Process underload fault';
	101:
		ErrorWord := 101;
		sErrorDescription := 'Process overload ';
	102:
		ErrorWord := 102;
		sErrorDescription := 'PI Feedback detectedfault'; 
	106:
		ErrorWord := 106;
		sErrorDescription := ' AI current lost fault ';
	
		
END_CASE
END_METHOD

METHOD StatusWord : E_InverterStatusWord
VAR_INPUT
	refMBdata : REFERENCE TO ARRAY[0..40] OF WORD;  //wskaźnik do tablicy ze słowem Controlnym 
END_VAR
// ETA Masked by 0x006F h -> Altivar modbus instructions


refMbdata[0] := refMBdata[0]  AND 16#006F;

CASE refMBdata[0] OF
	
	16#0028:
		StatusWord := eFaultDrive; // błąd komunikacja Modbus przerwana i nieaktywna
	16#0040: 
		StatusWord := eSwitchOnDisabled; // Stan po udanym resecie błędu komunikacji komedną eResetInv = 128
	16#0021: 
		StatusWord := eReadyToSwitchON; // Stan po ustawieniu gotowości Inverta komendą eReady = 14
	16#0023:
		StatusWord := eSwitchedOn; // Stan po ustawieniu komendy eFwd = 15 lub eRev = 2063 gdy jest zerowa prędkośc zadana speed = 0 
	16#0027:
		StatusWord := eOperationEnabled; // Stan gdy napęd pracuje w kierunku przodu po komendzie eFwd = 15 i osiągnał zadaną prędkość
	
		
END_CASE
END_METHOD

END_FUNCTION_BLOCK

// ---- POUs/Implementation/FB_DriveInverter.TcPOU
FUNCTION_BLOCK FB_DriveInverter EXTENDS FB_DriveReverse IMPLEMENTS I_DriveInverter;
VAR
	_stInverter : ST_Inverter;
			
END_VAR

VAR_STAT
	_nInstances		: INT;		// Counter of created Instances
END_VAR

PROPERTY DeviceData : ST_Inverter
GET
// Dane pobierane podczas obsługi Invertera przez ModbusRtu
DeviceData := _stInverter;
END_GET
SET
// Dane ustawiane podczas obsługi Invertera przez ModbusRtu
_stInverter := DeviceData;
END_SET
END_PROPERTY

METHOD FB_init : BOOL
VAR_INPUT
	bInitRetains : BOOL; // if TRUE, the retain variables are initialized (warm start / cold start)
	bInCopyCode : BOOL;  // if TRUE, the instance afterwards gets moved into the copy code (online change)
	bDeviceId		 : BYTE;	
END_VAR
THIS^._stInverter.bDeviceID := bDeviceID;

//count of FB Instances and setting int Array of Interface variables. Assign an object to an interface variable
// The array of interface variable must be global
_nInstances := _nInstances + 1;
Itf.aItfDriveInverter[_nInstances] := THIS^;
END_METHOD

PROPERTY InstanceCounter : INT
GET
InstanceCounter := _nInstances;
END_GET
END_PROPERTY

METHOD Reset : BOOL
VAR_INPUT
END_VAR

// Set reset Command
THIS^._eCommand := eResetInv;
END_METHOD

METHOD SetSpeed : BOOL
VAR_INPUT
	_speed	: REAL;
END_VAR
//Conversion speed to Inverter register Word 
THIS^._stInverter.rSpeed := REAL_TO_WORD(_speed * 10);
END_METHOD

METHOD StatusState :  E_StateDevice
VAR_INPUT
END_VAR
//Override 

// State Machine of the Drive 


CASE _eStateMachine OF
	
	eOff:
		WorkCounterOff();
		_supplyLed.State := FALSE;
		_stateLabel.Text := 'OFF';
		_statusLabel.Text := 'Napęd jest wyłączony';
		
		// Jesli falownik jest zasilony przejdz do stanu napęd w gotowości eOn
		IF _eCommand = eReady AND _termFuse.IsActive THEN
			_stInverter.eControl := eFaultReset;
			
			IF _stInverter.wStatus <> eFaultDrive AND _stInverter.wStatus <> eFaultAfterOperation THEN
				IF _stInverter.wStatus = eSwitchOnDisabled THEN
					_stInverter.eControl := eShutDown;
					
				END_IF
				
				IF _stInverter.wStatus = eReadyToSwitchOn THEN
					_stInverter.eControl := eSwitchOn;
					_eStateMachine := eOn;
				END_IF
	

			END_IF	
		END_IF
		
		
	
	eOn:
		WorkCounterOff();
		_supplyLed.State := TRUE;
		_stateLabel.Text := 'ON';
		_statusLabel.Text := 'Napęd jest w gotowości';

		// Uruchomienie napędu i przejscie do stanu eForward po potwierdzeniu slowa statusu eOperationEnabled
		IF _eCommand = eFwd THEN
			_stInverter.eControl := eEnableOperation;
			IF  _stInverter.wStatus = eOperationEnabled THEN
				_eStateMachine := eForward;
			END_IF
		// Uruchomienie napędu i przejscie do stanu eForward po potwierdzeniu slowa statusu eOperationEnabled
		ELSIF _eCommand = eRev THEN
			_stInverter.eControl := eReverseOperation;
			IF _stInverter.wStatus = eOperationEnabled THEN
				_eStateMachine := eReverse;
			END_IF
		END_IF 
		
        IF NOT _termFuse.IsActive THEN
			_eStateMachine := eOff;
		END_IF
		
		//Obsługa sytuacji blędu Modbusa przejdz do stanu eFault		
		IF _stInverter.errorMdb <> 0 THEN
 			_eStateMachine := eFault;
		END_IF
 
	
	eForward:
		_stateLabel.Text := 'RUNNING';
		_statusLabel.Text := 'Napęd jest uruchomiony do przodu';	
		WorkCounterOn();
		WorkCount();
		WorkTimelabel();	
		
		//Zatrzymaj napęd i przejdź do stanu gotowości eOn 
		IF _eCommand = eReady THEN 
			_stInverter.eControl := eSwitchOn;
			IF _stInverter.wStatus = eSwitchedOn THEN
				_eStateMachine := eOn;
			END_IF
		END_IF
		
		//Obsługa sytuacji zadziałania wyłacznika silnikowego przejdz do stanu eFault
        IF _eCommand = eFwd AND NOT _termFuse.IsActive THEN
			_eStateMachine := eFault;
		END_IF
		
		//Informacja o blędzie falownika 
		IF _stInverter.errorInv <> 0 THEN
			_statusLabel.Text := CONCAT('Błąd falownika nr:', WORD_TO_STRING(_stInverter.errorInv));
			_statusLabel.Text := CONCAT(_statuslabel.Text, _stInverter.sErrorDescription);
		END_IF
		
		//Obsługa sytuacji blędu Modbusa przejdz do stanu eFault
		IF _stInverter.errorMdb <> 0 THEN
 			_eStateMachine := eFault;
		END_IF
		
		//Jesli w Word Status Invertera jest status fault przejdz do stanu fault i zatrzymaj napęd
		IF _stInverter.wStatus = eFaultDrive OR _stInverter.wStatus =eFaultAfterOperation THEN
			_eStateMachine := eFault;
		END_IF
		
		
		
	eReverse:
		_stateLabel.Text := 'RUNNING';
		_statusLabel.Text := 'Napęd jest uruchomiony do tyłu';	
		WorkCounterOn();
		WorkCount();
		WorkTimelabel();
		IF _eCommand = eReady THEN
			_stInverter.eControl := eSwitchOn;
			IF _stInverter.wStatus = eSwitchedOn THEN
				_eStateMachine := eOn;
			END_IF
		END_IF
		
        IF _eCommand = eRev AND NOT _termFuse.IsActive THEN
			_eStateMachine := eFault;
		END_IF	
	 
		IF _stInverter.errorInv <> 0 THEN
			_statusLabel.Text := CONCAT('Błąd falownika nr:', WORD_TO_STRING(_stInverter.errorInv));
			_statusLabel.Text := CONCAT(_statuslabel.Text, _stInverter.sErrorDescription);
		END_IF
		
		IF _stInverter.errorMdb <> 0 THEN
 			_eStateMachine := eFault;
		END_IF
	

		IF _stInverter.wStatus = eFaultDrive OR _stInverter.wStatus =eFaultAfterOperation THEN
			_eStateMachine := eFault;
		END_IF
		
		
	eFault:
		//_stInverter.eControl := eSwitchOn;
		WorkCounterOff();
		_stateLabel.Text := 'FAULT';
		
		//wystąpił błąd falownika lub zadziałał wyłacznik silnikowy
		IF _termFuse.IsActive AND _stInverter.errorInv <> 0 THEN
			_statusLabel.Text := CONCAT('Błąd falownika nr:', WORD_TO_STRING(_stInverter.errorInv));
			_statusLabel.Text := CONCAT(_statuslabel.Text, _stInverter.sErrorDescription);
		ELSIF NOT _termFuse.IsActive THEN
			_statusLabel.Text := 'Zadziałał wyłacznik silnikowy';
		END_IF
		
		//wystąpił błąd Modbusa
		IF _stInverter.errorMdb <> 0 THEN
			_statusLabel.Text := CONCAT('Błąd sieci Modbus ', WORD_TO_STRING(_stInverter.errorMdb));
		END_IF		
		
		//wyłaczone zasilanie falownika przejdz do stanu eOff napęd wyłaczony
		IF _eCommand = eReady AND NOT _termFuse.IsActive THEN
			_eStateMachine := eOff;
		END_IF
			
		//wciśniety przycisk reset skasuj błąd falownika jesli się powiedzie przejdz do stanu eOff napęd wyłączony
		IF _eCommand = eResetInv THEN
			_stInverter.eControl := eFaultReset;
			IF  _stInverter.wStatus = eSwitchOnDisabled THEN 
				_statusLabel.Text := 'Bład falownika skasowany';
				_eStateMachine := eOff;
			END_IF
		END_IF

END_CASE
END_METHOD

METHOD SwitchOff : BOOL
VAR_INPUT
END_VAR
//Override  send "stop" command to modbus block
THIS^._eCommand := eReady;
END_METHOD

METHOD SwitchOn : BOOL
VAR_INPUT
END_VAR
//Override  send "start" command to Modbus block
THIS^._eCommand := eFwd;
END_METHOD

METHOD SwitchReverseOff : BOOL
//Override  send "reverse" stop command to Modbus block
THIS^._eCommand := eReady;
END_METHOD

METHOD SwitchReverseOn : BOOL
//Override  send "reverse" start command to Modbus block
THIS^._eCommand := eRev;
END_METHOD

END_FUNCTION_BLOCK

// ---- POUs/mergeIO.TcPOU
PROGRAM mergeIO
VAR
END_VAR


//Sygnały obiektów MccRev_* mieszadeł fermentora

//***************************************************SCADA********************************************************

////MccRev_001 variable sets by SCADA
//FermentationProcess.fbMccRev_001.ScadaAutoButton     := MccRev_001.bAutoButton;    // SCADA button Auto Command
//FermentationProcess.fbMccRev_001.ScadaForwardButton  := MccRev_001.bForwardButton; // SCADA button Forward Command
//FermentationProcess.fbMccRev_001.ScadaReverseButton  := MccRev_001.bReverseButton; // SCADA button Reverse Command

////MccRev_002 variable sets by SCADA
//FermentationProcess.fbMccRev_002.ScadaAutoButton     := MccRev_002.bAutoButton;    // SCADA button Auto Command
//FermentationProcess.fbMccRev_002.ScadaForwardButton  := MccRev_002.bForwardButton; // SCADA button Forward Command
//FermentationProcess.fbMccRev_002.ScadaReverseButton  := MccRev_002.bReverseButton; // SCADA button Reverse Command

////MccRev_003 variable sets by SCADA
//FermentationProcess.fbMccRev_003.ScadaAutoButton     := MccRev_003.bAutoButton;    // SCADA button Auto Command
//FermentationProcess.fbMccRev_003.ScadaForwardButton  := MccRev_003.bForwardButton; // SCADA button Forward Command
//FermentationProcess.fbMccRev_003.ScadaReverseButton  := MccRev_003.bReverseButton; // SCADA button Reverse Command

////MccRev_004 variable sets by SCADA
//FermentationProcess.fbMccRev_004.ScadaAutoButton     := MccRev_004.bAutoButton;    // SCADA button Auto Command
//FermentationProcess.fbMccRev_004.ScadaForwardButton  := MccRev_004.bForwardButton; // SCADA button Forward Command
//FermentationProcess.fbMccRev_004.ScadaReverseButton  := MccRev_004.bReverseButton; // SCADA button Reverse Command

////MccRev_005 variable sets by SCADA
//FermentationProcess.fbMccRev_005.ScadaAutoButton     := MccRev_005.bAutoButton;    // SCADA button Auto Command
//FermentationProcess.fbMccRev_005.ScadaForwardButton  := MccRev_005.bForwardButton; // SCADA button Forward Command
//FermentationProcess.fbMccRev_005.ScadaReverseButton  := MccRev_005.bReverseButton; // SCADA button Reverse Command

////MccRev_006 variable sets by SCADA
//FermentationProcess.fbMccRev_006.ScadaAutoButton     := MccRev_006.bAutoButton;    // SCADA button Auto Command
//FermentationProcess.fbMccRev_006.ScadaForwardButton  := MccRev_006.bForwardButton; // SCADA button Forward Command
//FermentationProcess.fbMccRev_006.ScadaReverseButton  := MccRev_006.bReverseButton; // SCADA button Reverse Command

////MccRev_007 variable sets by SCADA
//FermentationProcess.fbMccRev_007.ScadaAutoButton     := MccRev_007.bAutoButton;    // SCADA button Auto Command
//FermentationProcess.fbMccRev_007.ScadaForwardButton  := MccRev_007.bForwardButton; // SCADA button Forward Command
//FermentationProcess.fbMccRev_007.ScadaReverseButton  := MccRev_007.bReverseButton; // SCADA button Reverse Command

////MccRev_008 variable sets by SCADA
//FermentationProcess.fbMccRev_008.ScadaAutoButton     := MccRev_008.bAutoButton;    // SCADA button Auto Command
//FermentationProcess.fbMccRev_008.ScadaForwardButton  := MccRev_008.bForwardButton; // SCADA button Forward Command
//FermentationProcess.fbMccRev_008.ScadaReverseButton  := MccRev_008.bReverseButton; // SCADA button Reverse Command

////MccRev_009 variable sets by SCADA
//FermentationProcess.fbMccRev_009.ScadaAutoButton     := MccRev_009.bAutoButton;    // SCADA button Auto Command
//FermentationProcess.fbMccRev_009.ScadaForwardButton  := MccRev_009.bForwardButton; // SCADA button Forward Command
//FermentationProcess.fbMccRev_009.ScadaReverseButton  := MccRev_009.bReverseButton; // SCADA button Reverse Command

////MccRev_010 variable sets by SCADA
//FermentationProcess.fbMccRev_010.ScadaAutoButton     := MccRev_010.bAutoButton;    // SCADA button Auto Command
//FermentationProcess.fbMccRev_010.ScadaForwardButton  := MccRev_010.bForwardButton; // SCADA button Forward Command
//FermentationProcess.fbMccRev_010.ScadaReverseButton  := MccRev_010.bReverseButton; // SCADA button Reverse Command

////MccRev_011 variable sets by SCADA
//FermentationProcess.fbMccRev_011.ScadaAutoButton     := MccRev_011.bAutoButton;    // SCADA button Auto Command
//FermentationProcess.fbMccRev_011.ScadaForwardButton  := MccRev_011.bForwardButton; // SCADA button Forward Command
//FermentationProcess.fbMccRev_011.ScadaReverseButton  := MccRev_011.bReverseButton; // SCADA button Reverse Command

////MccRev_012 variable sets by SCADA
//FermentationProcess.fbMccRev_012.ScadaAutoButton     := MccRev_012.bAutoButton;    // SCADA button Auto Command
//FermentationProcess.fbMccRev_012.ScadaForwardButton  := MccRev_012.bForwardButton; // SCADA button Forward Command
//FermentationProcess.fbMccRev_012.ScadaReverseButton  := MccRev_012.bReverseButton; // SCADA button Reverse Command

////MccRev_013 variable sets by SCADA
//FermentationProcess.fbMccRev_013.ScadaAutoButton     := MccRev_013.bAutoButton;    // SCADA button Auto Command
//FermentationProcess.fbMccRev_013.ScadaForwardButton  := MccRev_013.bForwardButton; // SCADA button Forward Command
//FermentationProcess.fbMccRev_013.ScadaReverseButton  := MccRev_013.bReverseButton; // SCADA button Reverse Command

////MccRev_014 variable sets by SCADA
//FermentationProcess.fbMccRev_014.ScadaAutoButton     := MccRev_014.bAutoButton;    // SCADA button Auto Command
//FermentationProcess.fbMccRev_014.ScadaForwardButton  := MccRev_014.bForwardButton; // SCADA button Forward Command
//FermentationProcess.fbMccRev_014.ScadaReverseButton  := MccRev_014.bReverseButton; // SCADA button Reverse Command

////MccRev_015 variable sets by SCADA
//FermentationProcess.fbMccRev_015.ScadaAutoButton     := MccRev_015.bAutoButton;    // SCADA button Auto Command
//FermentationProcess.fbMccRev_015.ScadaForwardButton  := MccRev_015.bForwardButton; // SCADA button Forward Command
//FermentationProcess.fbMccRev_015.ScadaReverseButton  := MccRev_015.bReverseButton; // SCADA button Reverse Command

////MccRev_016 variable sets by SCADA
//FermentationProcess.fbMccRev_016.ScadaAutoButton     := MccRev_016.bAutoButton;    // SCADA button Auto Command
//FermentationProcess.fbMccRev_016.ScadaForwardButton  := MccRev_016.bForwardButton; // SCADA button Forward Command
//FermentationProcess.fbMccRev_016.ScadaReverseButton  := MccRev_016.bReverseButton; // SCADA button Reverse Command

////MccRev_017 variable sets by SCADA
//FermentationProcess.fbMccRev_017.ScadaAutoButton     := MccRev_017.bAutoButton;    // SCADA button Auto Command
//FermentationProcess.fbMccRev_017.ScadaForwardButton  := MccRev_017.bForwardButton; // SCADA button Forward Command
//FermentationProcess.fbMccRev_017.ScadaReverseButton  := MccRev_017.bReverseButton; // SCADA button Reverse Command

////MccRev_018 variable sets by SCADA
//FermentationProcess.fbMccRev_018.ScadaAutoButton     := MccRev_018.bAutoButton;    // SCADA button Auto Command
//FermentationProcess.fbMccRev_018.ScadaForwardButton  := MccRev_018.bForwardButton; // SCADA button Forward Command
//FermentationProcess.fbMccRev_018.ScadaReverseButton  := MccRev_018.bReverseButton; // SCADA button Reverse Command

////MccRev_019 variable sets by SCADA
//FermentationProcess.fbMccRev_019.ScadaAutoButton     := MccRev_019.bAutoButton;    // SCADA button Auto Command
//FermentationProcess.fbMccRev_019.ScadaForwardButton  := MccRev_019.bForwardButton; // SCADA button Forward Command
//FermentationProcess.fbMccRev_019.ScadaReverseButton  := MccRev_019.bReverseButton; // SCADA button Reverse Command

////MccRev_020 variable sets by SCADA
//FermentationProcess.fbMccRev_020.ScadaAutoButton     := MccRev_020.bAutoButton;    // SCADA button Auto Command
//FermentationProcess.fbMccRev_020.ScadaForwardButton  := MccRev_020.bForwardButton; // SCADA button Forward Command
//FermentationProcess.fbMccRev_020.ScadaReverseButton  := MccRev_020.bReverseButton; // SCADA button Reverse Command


////***************************************************PLC********************************************************************


////MccRev_001 variable sets by PLC
//MccRev_001.bTermFuse      := FermentationProcess.fbDriveReverse_001.MotorProtection;  // PLC input thermal fuse
//MccRev_001.bContactor     := FermentationProcess.fbDriveReverse_001.MotorContactor;   // PLC output contactor
//MccRev_001.udHours        := FermentationProcess.fbDriveReverse_001.Hours;            // PLC Work Time Counter - hours nonvolatile memory register
//MccRev_001.uMinutes       := FermentationProcess.fbDriveReverse_001.Minuts;           // PLC Work Time Counter - minutes nonvolatile memory register
//MccRev_001.uSeconds       := FermentationProcess.fbDriveReverse_001.Seconds;          // PLC Work Time Counter - seconds nonvolatile memory register
//MccRev_001.sState         := FermentationProcess.fbDriveReverse_001.MotorState;       // PLC Work Time Counter - minutes nonvolatile memory register
//MccRev_001.sStatus        := FermentationProcess.fbDriveReverse_001.MotorStatus;      // PLC Work Time Counter - seconds nonvolatile memory register


////MccRev_002 variable sets by PLC
//MccRev_002.bTermFuse      := FermentationProcess.fbDriveReverse_002.MotorProtection;  // PLC input thermal fuse
//MccRev_002.bContactor     := FermentationProcess.fbDriveReverse_002.MotorContactor;   // PLC output contactor
//MccRev_002.udHours        := FermentationProcess.fbDriveReverse_002.Hours;            // PLC Work Time Counter - hours nonvolatile memory register
//MccRev_002.uMinutes       := FermentationProcess.fbDriveReverse_002.Minuts;           // PLC Work Time Counter - minutes nonvolatile memory register
//MccRev_002.uSeconds       := FermentationProcess.fbDriveReverse_002.Seconds;          // PLC Work Time Counter - seconds nonvolatile memory register
//MccRev_002.sState         := FermentationProcess.fbDriveReverse_002.MotorState;       // PLC Work Time Counter - minutes nonvolatile memory register
//MccRev_002.sStatus        := FermentationProcess.fbDriveReverse_002.MotorStatus;      // PLC Work Time Counter - seconds nonvolatile memory register

////MccRev_003 variable sets by PLC
//MccRev_003.bTermFuse      := FermentationProcess.fbDriveReverse_003.MotorProtection;  // PLC input thermal fuse
//MccRev_003.bContactor     := FermentationProcess.fbDriveReverse_003.MotorContactor;   // PLC output contactor
//MccRev_003.udHours        := FermentationProcess.fbDriveReverse_003.Hours;            // PLC Work Time Counter - hours nonvolatile memory register
//MccRev_003.uMinutes       := FermentationProcess.fbDriveReverse_003.Minuts;           // PLC Work Time Counter - minutes nonvolatile memory register
//MccRev_003.uSeconds       := FermentationProcess.fbDriveReverse_003.Seconds;          // PLC Work Time Counter - seconds nonvolatile memory register
//MccRev_003.sState         := FermentationProcess.fbDriveReverse_003.MotorState;       // PLC Work Time Counter - minutes nonvolatile memory register
//MccRev_003.sStatus        := FermentationProcess.fbDriveReverse_003.MotorStatus;      // PLC Work Time Counter - seconds nonvolatile memory register

////MccRev_004 variable sets by PLC
//MccRev_004.bTermFuse      := FermentationProcess.fbDriveReverse_004.MotorProtection;  // PLC input thermal fuse
//MccRev_004.bContactor     := FermentationProcess.fbDriveReverse_004.MotorContactor;   // PLC output contactor
//MccRev_004.udHours        := FermentationProcess.fbDriveReverse_004.Hours;            // PLC Work Time Counter - hours nonvolatile memory register
//MccRev_004.uMinutes       := FermentationProcess.fbDriveReverse_004.Minuts;           // PLC Work Time Counter - minutes nonvolatile memory register
//MccRev_004.uSeconds       := FermentationProcess.fbDriveReverse_004.Seconds;          // PLC Work Time Counter - seconds nonvolatile memory register
//MccRev_004.sState         := FermentationProcess.fbDriveReverse_004.MotorState;       // PLC Work Time Counter - minutes nonvolatile memory register
//MccRev_004.sStatus        := FermentationProcess.fbDriveReverse_004.MotorStatus;      // PLC Work Time Counter - seconds nonvolatile memory register


